RoboDK station: kr30 cnc template half inch flat end mill - paulina 4 AAAAAAAAAAAAAAAAAAAA.rdk

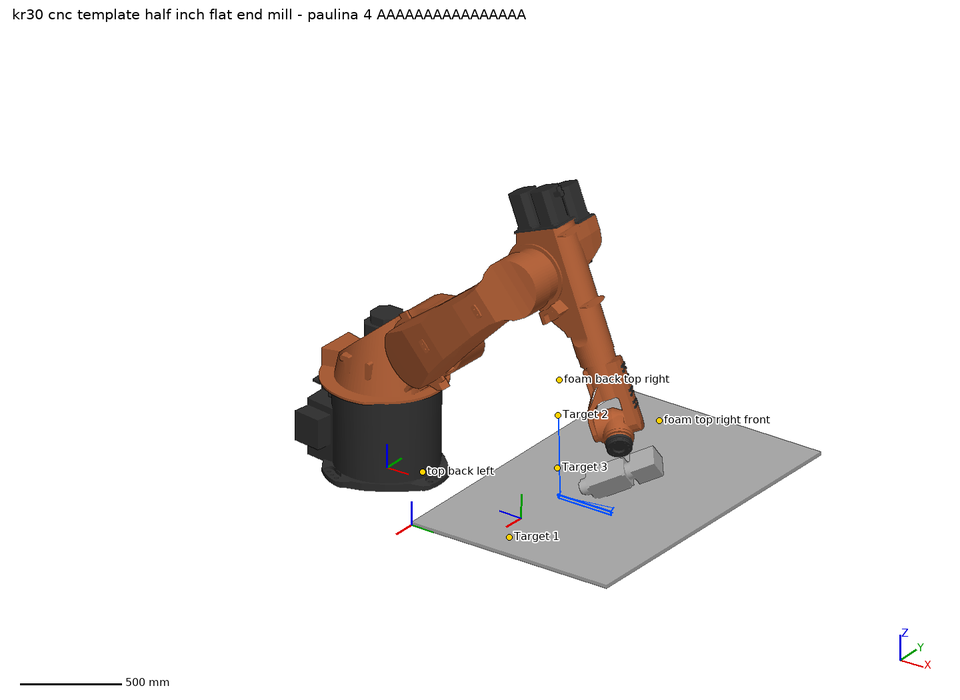
[picture v0: the station drawn from its stored meshes, robots at their saved joint values, targets as dots, program paths as lines]
Station kr30 cnc template half inch flat end mill - paulina 4 AAAAAAAAAAAAAAAAAAAA. Poses are relative to the parent item; angles as X-Y-Z fixed-axis rotations.
  - frame KUKA KR 30 HA Base at (0, 0, 0) mm
    - robot KUKA KR 30 HA: 6 axes, payload 30 kg, reach 2033 mm, repeatability 0.05 mm, weight 665 kg
        modified DH rows (alpha deg, a mm, theta deg, d mm): 0, 0, 0, 815; -90, 350, 0, 0; 0, 850, -90, 0; -90, 145, 0, 820; 90, 0, 0, 0; -90, 0, 180, 170
        joint limits [-185, -135, -120, -350, -119, -350] to [185, 35, 158, 350, 119, 350]; home [0, -90, 90, 0, 0, 0]; saved at [2.296, -41.464, 109.826, -239.674, 53.216, 262.884]
      - tool rc90 spindle mm, TCP at (337.31, -2.2, 160.57) mm, size 110 x 421.3 x 118 mm, geometry from rc90 spindle mm.stl
    - frame Tabletop at (921.82, -1104.91, 385) mm, rotated rx -0.93 ry -0.21 rz -89.9 deg
      - object tabletop CHECK HEIGHT at (-1839.9, 0, 0) mm, size 1839.9 x 1168.4 x 19 mm, geometry from kr30 tabletop mm.stl
      - object kr30 pipe jig base at (-1220, -610.6, 0) mm, size 1217.6 x 88.9 x 88.9 mm, geometry from kr30 pipe jig base.stl
      - frame Frame 3 at (-340, 420, 29) mm, rotated rx 90 ry 0 rz 0 deg
        - target Target 1 (Cartesian target) at (324.46, 69.12, -153.95) mm, rotated rx -179.9 ry 0.14 rz -89.96 deg; joints [37.245, -66.694, 101.534, 53.768, -48.608, -41.204] of KUKA KR 30 HA
        - target Target 2 (Cartesian target) at (-319.2, 432.53, 9.87) mm, rotated rx -179.07 ry 0.05 rz -32.45 deg; joints [8.715, -80.767, 140.791, -170.364, 60.256, 232.965] of KUKA KR 30 HA
        - target Target 3 (Cartesian target) at (-219.35, 204.08, -59.86) mm, rotated rx -178.17 ry 0.56 rz -29.88 deg; joints [13.008, -58.669, 136.899, -167.101, 79.453, 237.713] of KUKA KR 30 HA
    - target foam back top right (Cartesian target) at (1197.65, -230.62, 906.79) mm, rotated rx -15.53 ry 90 rz -15.53 deg; joints [14.757, -102.447, 141.256, 22.791, -41.102, -17.568] of KUKA KR 30 HA
    - target foam top right front (Cartesian target) at (1797.45, -230.62, 850.68) mm, rotated rx -15.58 ry 90 rz -15.58 deg; joints [8.85, -62.405, 99.608, 14.434, -38.093, -11.451] of KUKA KR 30 HA
    - target top back left (Cartesian target) at (1223.08, -1440.01, 894.96) mm, rotated rx 58.97 ry 90 rz 58.97 deg; joints [58.171, -50.232, 76.73, 74.515, -61.834, -59.599] of KUKA KR 30 HA
  - machining project Machining Settings: C:/Users/Research Office/Downloads/b4.apt | rotZ(0) | rotX(0)*rotY(0) | roty(-35) | onStart | onPathStart | onApproach | onPoint | onRetract | onFinish | SetTool(%1) | onPathFinish
  - program Machining (294 instructions, listed below)
  - program Machining (293 instructions, listed below)
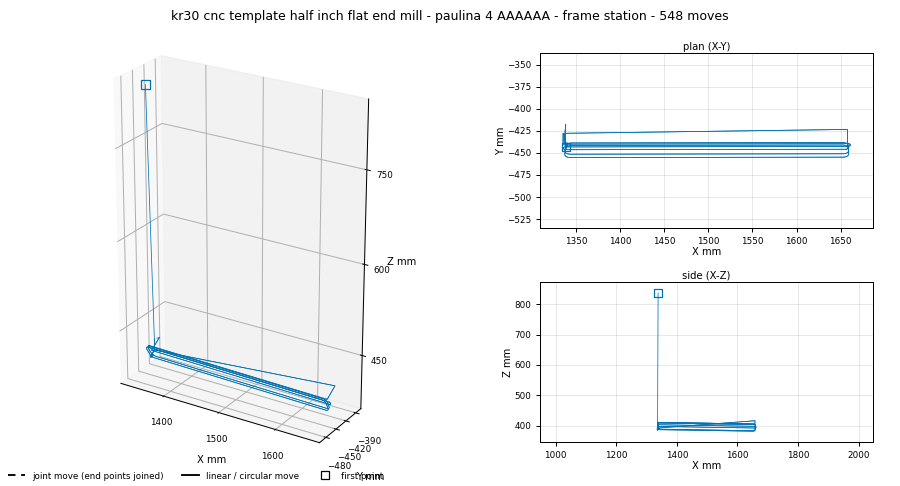
[picture p0: tool path of kr30 cnc template half inch flat end mill - paulina 4 AAAAAAAAAAAAAAAAAAAA.rdk in frame station, 548 of 548 moves have a stored position in this frame; points joined in program order, loops and branches not executed]

--- program Machining (robot KUKA KR 30 HA) ---
  Smooth(10)
  Print: /'1001'
  Print: /''
  Print: /'Contour3'
  Call SetTool(1)
  Set speed (200.0 mm/s)
  Set Ref.: Frame 3
  Set Tool: rc90 spindle mm
  Show rc90 spindle mm
  Set speed (200.0 mm/s)
  MoveJ (Target 2)
  MoveL 619 to (-335.6, -11.85, 4.35) mm, rotated rx -179.15 ry 0 rz -30.08 deg; joints [7.518, -42.725, 139.823, -172.763, 96.85, 241.025]
  MoveL 620 to (-332.9, -13.41, 4.35) mm, rotated rx -179.15 ry 0 rz -30.08 deg; joints [7.669, -42.588, 139.757, -172.61, 96.919, 241.053]
  Set speed (50.0 mm/s)
  MoveL 621 to (-326.98, -16.84, 4.35) mm, rotated rx -179.15 ry 0 rz -30.08 deg; joints [8, -42.287, 139.611, -172.274, 97.068, 241.115]
  MoveL 622 to (-325.36, -16.57, 3.64) mm, rotated rx -179.15 ry 0 rz -30.08 deg; joints [8.085, -42.306, 139.552, -172.19, 96.989, 241.115]
  Set speed (100.0 mm/s)
  MoveL 623 to (-324.39, -14.89, 2.31) mm, rotated rx -179.15 ry 0 rz -30.08 deg; joints [8.128, -42.444, 139.493, -172.15, 96.793, 241.093]
  MoveC 624 to (-324.11, -14.42, 1.33) mm, rotated rx -179.15 ry 0 rz -30.08 deg; joints [8.135, -42.479, 139.434, -172.144, 96.699, 241.081] to (-324.33, -14.8, 0.3) mm, rotated rx -179.15 ry 0 rz -30.08 deg; joints [8.115, -42.44, 139.354, -172.165, 96.659, 241.073]
  MoveL 625 to (-324.33, -14.8, 0.3) mm, rotated rx -179.15 ry 0 rz -30.08 deg; joints [8.115, -42.44, 139.354, -172.165, 96.659, 241.073]
  MoveL 626 to (-324.51, -15.11, -0.05) mm, rotated rx -179.15 ry 0 rz -30.08 deg; joints [8.102, -42.411, 139.324, -172.178, 96.658, 241.071]
  MoveL 627 to (-324.67, -15.38, -0.39) mm, rotated rx -179.15 ry 0 rz -30.08 deg; joints [8.091, -42.385, 139.294, -172.189, 96.654, 241.07]
  MoveL 628 to (-324.81, -15.61, -0.73) mm, rotated rx -179.15 ry 0 rz -30.08 deg; joints [8.081, -42.363, 139.266, -172.2, 96.648, 241.067]
  MoveL 629 to (-324.92, -15.82, -1.07) mm, rotated rx -179.15 ry 0 rz -30.08 deg; joints [8.071, -42.343, 139.237, -172.209, 96.64, 241.065]
  MoveL 630 to (-325.03, -15.99, -1.42) mm, rotated rx -179.15 ry 0 rz -30.08 deg; joints [8.063, -42.326, 139.21, -172.218, 96.63, 241.063]
  MoveL 631 to (-325.11, -16.15, -1.76) mm, rotated rx -179.15 ry 0 rz -30.08 deg; joints [8.055, -42.311, 139.183, -172.225, 96.618, 241.06]
  MoveL 632 to (-325.19, -16.28, -2.1) mm, rotated rx -179.15 ry 0 rz -30.08 deg; joints [8.049, -42.297, 139.156, -172.232, 96.605, 241.058]
  MoveL 633 to (-325.25, -16.39, -2.45) mm, rotated rx -179.15 ry 0 rz -30.08 deg; joints [8.042, -42.285, 139.13, -172.239, 96.591, 241.055]
  MoveL 634 to (-325.31, -16.48, -2.8) mm, rotated rx -179.15 ry 0 rz -30.08 deg; joints [8.037, -42.275, 139.103, -172.245, 96.575, 241.052]
  MoveL 635 to (-325.35, -16.55, -3.14) mm, rotated rx -179.15 ry 0 rz -30.08 deg; joints [8.032, -42.267, 139.077, -172.25, 96.558, 241.049]
  MoveL 636 to (-325.38, -16.61, -3.49) mm, rotated rx -179.15 ry 0 rz -30.08 deg; joints [8.027, -42.26, 139.052, -172.255, 96.54, 241.046]
  MoveL 637 to (-325.41, -16.65, -3.84) mm, rotated rx -179.15 ry 0 rz -30.08 deg; joints [8.023, -42.254, 139.026, -172.26, 96.52, 241.043]
  MoveL 638 to (-325.42, -16.67, -4.19) mm, rotated rx -179.15 ry 0 rz -30.08 deg; joints [8.02, -42.25, 139.001, -172.263, 96.499, 241.04]
  MoveL 639 to (-325.42, -16.68, -4.54) mm, rotated rx -179.15 ry 0 rz -30.08 deg; joints [8.017, -42.247, 138.977, -172.267, 96.478, 241.036]
  MoveL 640 to (-325.42, -16.68, -311.19) mm, rotated rx -179.15 ry 0 rz -30.08 deg; joints [6.155, -36.963, 115.713, -174.061, 78.617, 238.976]
  MoveL 641 to (-325.42, -16.67, -311.54) mm, rotated rx -179.15 ry 0 rz -30.08 deg; joints [6.154, -36.954, 115.684, -174.062, 78.597, 238.974]
  MoveL 642 to (-325.41, -16.65, -311.88) mm, rotated rx -179.15 ry 0 rz -30.08 deg; joints [6.152, -36.946, 115.655, -174.062, 78.577, 238.972]
  MoveL 643 to (-325.38, -16.61, -312.23) mm, rotated rx -179.15 ry 0 rz -30.08 deg; joints [6.152, -36.94, 115.627, -174.063, 78.556, 238.97]
  MoveL 644 to (-325.35, -16.55, -312.58) mm, rotated rx -179.15 ry 0 rz -30.08 deg; joints [6.152, -36.934, 115.599, -174.062, 78.533, 238.968]
  MoveL 645 to (-325.31, -16.48, -312.93) mm, rotated rx -179.15 ry 0 rz -30.08 deg; joints [6.152, -36.93, 115.572, -174.062, 78.51, 238.965]
  MoveL 646 to (-325.25, -16.39, -313.28) mm, rotated rx -179.15 ry 0 rz -30.08 deg; joints [6.152, -36.926, 115.544, -174.061, 78.486, 238.963]
  MoveL 647 to (-325.19, -16.27, -313.63) mm, rotated rx -179.15 ry 0 rz -30.08 deg; joints [6.154, -36.924, 115.517, -174.059, 78.462, 238.96]
  MoveL 648 to (-325.11, -16.14, -313.98) mm, rotated rx -179.15 ry 0 rz -30.08 deg; joints [6.155, -36.923, 115.491, -174.057, 78.436, 238.957]
  MoveL 649 to (-325.02, -15.98, -314.33) mm, rotated rx -179.15 ry 0 rz -30.08 deg; joints [6.157, -36.924, 115.464, -174.054, 78.409, 238.953]
  MoveL 650 to (-324.91, -15.8, -314.68) mm, rotated rx -179.15 ry 0 rz -30.08 deg; joints [6.16, -36.926, 115.438, -174.05, 78.381, 238.95]
  MoveL 651 to (-324.79, -15.59, -315.03) mm, rotated rx -179.15 ry 0 rz -30.08 deg; joints [6.164, -36.93, 115.413, -174.046, 78.352, 238.946]
  MoveL 652 to (-324.65, -15.35, -315.38) mm, rotated rx -179.15 ry 0 rz -30.08 deg; joints [6.168, -36.936, 115.388, -174.041, 78.321, 238.942]
  MoveL 653 to (-324.5, -15.09, -315.7) mm, rotated rx -179.15 ry 0 rz -30.08 deg; joints [6.173, -36.944, 115.365, -174.036, 78.291, 238.938]
  MoveL 654 to (-324.33, -14.8, -316.02) mm, rotated rx -179.15 ry 0 rz -30.08 deg; joints [6.179, -36.954, 115.343, -174.029, 78.259, 238.933]
  MoveL 655 to (-324.16, -14.49, -316.3) mm, rotated rx -179.15 ry 0 rz -30.08 deg; joints [6.185, -36.965, 115.325, -174.022, 78.229, 238.929]
  MoveL 656 to (-323.98, -14.19, -316.55) mm, rotated rx -179.15 ry 0 rz -30.08 deg; joints [6.191, -36.978, 115.309, -174.015, 78.202, 238.924]
  MoveL 657 to (-323.81, -13.89, -316.76) mm, rotated rx -179.15 ry 0 rz -30.08 deg; joints [6.197, -36.991, 115.296, -174.008, 78.176, 238.92]
  MoveL 658 to (-323.63, -13.59, -316.94) mm, rotated rx -179.15 ry 0 rz -30.08 deg; joints [6.204, -37.005, 115.286, -174.001, 78.151, 238.916]
  MoveL 659 to (-323.46, -13.29, -317.1) mm, rotated rx -179.15 ry 0 rz -30.08 deg; joints [6.21, -37.02, 115.277, -173.994, 78.129, 238.913]
  MoveL 660 to (-323.28, -12.99, -317.23) mm, rotated rx -179.15 ry 0 rz -30.08 deg; joints [6.217, -37.036, 115.271, -173.986, 78.107, 238.909]
  MoveL 661 to (-323.11, -12.68, -317.34) mm, rotated rx -179.15 ry 0 rz -30.08 deg; joints [6.224, -37.052, 115.266, -173.979, 78.087, 238.905]
  MoveL 662 to (-322.93, -12.38, -317.43) mm, rotated rx -179.15 ry 0 rz -30.08 deg; joints [6.231, -37.068, 115.264, -173.971, 78.068, 238.902]
  MoveL 663 to (-322.76, -12.08, -317.5) mm, rotated rx -179.15 ry 0 rz -30.08 deg; joints [6.238, -37.085, 115.263, -173.964, 78.05, 238.898]
  MoveL 664 to (-322.58, -11.78, -317.55) mm, rotated rx -179.15 ry 0 rz -30.08 deg; joints [6.245, -37.103, 115.263, -173.956, 78.033, 238.895]
  MoveL 665 to (-322.41, -11.48, -317.58) mm, rotated rx -179.15 ry 0 rz -30.08 deg; joints [6.252, -37.121, 115.266, -173.948, 78.017, 238.892]
  MoveL 666 to (-322.23, -11.17, -317.59) mm, rotated rx -179.15 ry 0 rz -30.08 deg; joints [6.26, -37.14, 115.27, -173.94, 78.003, 238.889]
  MoveL 667 to (-315.94, -0.31, -317.59) mm, rotated rx -179.15 ry 0 rz -30.08 deg; joints [6.525, -37.821, 115.428, -173.657, 77.489, 238.774]
  MoveL 668 to (-315.59, 0.29, -317.58) mm, rotated rx -179.15 ry 0 rz -30.08 deg; joints [6.54, -37.859, 115.438, -173.641, 77.461, 238.768]
  MoveL 669 to (-315.42, 0.6, -317.55) mm, rotated rx -179.15 ry 0 rz -30.08 deg; joints [6.547, -37.879, 115.444, -173.633, 77.448, 238.765]
  MoveL 670 to (-315.24, 0.9, -317.5) mm, rotated rx -179.15 ry 0 rz -30.08 deg; joints [6.555, -37.899, 115.452, -173.625, 77.437, 238.762]
  MoveL 671 to (-315.07, 1.2, -317.43) mm, rotated rx -179.15 ry 0 rz -30.08 deg; joints [6.562, -37.92, 115.462, -173.617, 77.426, 238.759]
  MoveL 672 to (-314.89, 1.5, -317.34) mm, rotated rx -179.15 ry 0 rz -30.08 deg; joints [6.57, -37.941, 115.474, -173.609, 77.416, 238.756]
  MoveL 673 to (-314.72, 1.8, -317.23) mm, rotated rx -179.15 ry 0 rz -30.08 deg; joints [6.578, -37.963, 115.487, -173.6, 77.408, 238.753]
  MoveL 674 to (-314.54, 2.1, -317.1) mm, rotated rx -179.15 ry 0 rz -30.08 deg; joints [6.586, -37.986, 115.502, -173.592, 77.401, 238.75]
  MoveL 675 to (-314.39, 2.36, -316.97) mm, rotated rx -179.15 ry 0 rz -30.08 deg; joints [6.593, -38.005, 115.517, -173.585, 77.396, 238.748]
  MoveL 676 to (-314.24, 2.62, -316.82) mm, rotated rx -179.15 ry 0 rz -30.08 deg; joints [6.6, -38.026, 115.533, -173.577, 77.392, 238.746]
  MoveL 677 to (-314.09, 2.88, -316.65) mm, rotated rx -179.15 ry 0 rz -30.08 deg; joints [6.607, -38.047, 115.551, -173.57, 77.389, 238.744]
  MoveL 678 to (-313.95, 3.13, -316.45) mm, rotated rx -179.15 ry 0 rz -30.08 deg; joints [6.614, -38.068, 115.57, -173.563, 77.387, 238.743]
  MoveL 679 to (-313.8, 3.39, -316.23) mm, rotated rx -179.15 ry 0 rz -30.08 deg; joints [6.622, -38.09, 115.592, -173.555, 77.387, 238.741]
  MoveL 680 to (-313.65, 3.65, -315.98) mm, rotated rx -179.15 ry 0 rz -30.08 deg; joints [6.629, -38.113, 115.616, -173.547, 77.388, 238.739]
  MoveL 681 to (-313.49, 3.92, -315.68) mm, rotated rx -179.15 ry 0 rz -30.08 deg; joints [6.638, -38.139, 115.645, -173.539, 77.392, 238.738]
  MoveL 682 to (-313.35, 4.16, -315.38) mm, rotated rx -179.15 ry 0 rz -30.08 deg; joints [6.645, -38.162, 115.673, -173.532, 77.397, 238.737]
  MoveL 683 to (-313.24, 4.35, -315.11) mm, rotated rx -179.15 ry 0 rz -30.08 deg; joints [6.651, -38.181, 115.698, -173.526, 77.402, 238.736]
  MoveL 684 to (-313.14, 4.52, -314.85) mm, rotated rx -179.15 ry 0 rz -30.08 deg; joints [6.656, -38.199, 115.722, -173.52, 77.409, 238.736]
  MoveL 685 to (-313.05, 4.68, -314.57) mm, rotated rx -179.15 ry 0 rz -30.08 deg; joints [6.662, -38.217, 115.747, -173.515, 77.416, 238.735]
  MoveL 686 to (-312.97, 4.82, -314.28) mm, rotated rx -179.15 ry 0 rz -30.08 deg; joints [6.666, -38.234, 115.773, -173.51, 77.425, 238.735]
  MoveL 687 to (-312.9, 4.95, -314) mm, rotated rx -179.15 ry 0 rz -30.08 deg; joints [6.671, -38.249, 115.798, -173.506, 77.435, 238.735]
  MoveL 688 to (-312.83, 5.06, -313.72) mm, rotated rx -179.15 ry 0 rz -30.08 deg; joints [6.675, -38.264, 115.823, -173.502, 77.445, 238.736]
  MoveL 689 to (-312.73, 5.24, -313.15) mm, rotated rx -179.15 ry 0 rz -30.08 deg; joints [6.682, -38.291, 115.872, -173.495, 77.467, 238.737]
  MoveL 690 to (-312.65, 5.37, -312.58) mm, rotated rx -179.15 ry 0 rz -30.08 deg; joints [6.688, -38.315, 115.92, -173.489, 77.492, 238.738]
  MoveL 691 to (-312.62, 5.43, -312.23) mm, rotated rx -179.15 ry 0 rz -30.08 deg; joints [6.692, -38.328, 115.95, -173.486, 77.508, 238.739]
  MoveL 692 to (-312.59, 5.47, -311.88) mm, rotated rx -179.15 ry 0 rz -30.08 deg; joints [6.694, -38.34, 115.979, -173.484, 77.525, 238.741]
  MoveL 693 to (-312.58, 5.49, -311.54) mm, rotated rx -179.15 ry 0 rz -30.08 deg; joints [6.697, -38.351, 116.009, -173.482, 77.543, 238.742]
  MoveL 694 to (-312.58, 5.49, -311.19) mm, rotated rx -179.15 ry 0 rz -30.08 deg; joints [6.699, -38.361, 116.037, -173.481, 77.562, 238.744]
  MoveL 695 to (-312.58, 5.49, -5.24) mm, rotated rx -179.15 ry 0 rz -30.08 deg; joints [8.711, -44.154, 139.346, -171.59, 94.945, 240.891]
  MoveL 696 to (-312.58, 5.49, -2.45) mm, rotated rx -179.15 ry 0 rz -30.08 deg; joints [8.735, -44.177, 139.543, -171.564, 95.117, 240.919]
  MoveL 697 to (-312.59, 5.47, -2.1) mm, rotated rx -179.15 ry 0 rz -30.08 deg; joints [8.737, -44.178, 139.568, -171.562, 95.14, 240.923]
  MoveL 698 to (-312.62, 5.43, -1.75) mm, rotated rx -179.15 ry 0 rz -30.08 deg; joints [8.739, -44.178, 139.592, -171.56, 95.164, 240.926]
  MoveL 699 to (-312.65, 5.37, -1.4) mm, rotated rx -179.15 ry 0 rz -30.08 deg; joints [8.74, -44.176, 139.615, -171.558, 95.19, 240.93]
  MoveL 700 to (-312.69, 5.3, -1.05) mm, rotated rx -179.15 ry 0 rz -30.08 deg; joints [8.741, -44.172, 139.639, -171.557, 95.216, 240.934]
  MoveL 701 to (-312.75, 5.2, -0.7) mm, rotated rx -179.15 ry 0 rz -30.08 deg; joints [8.741, -44.167, 139.662, -171.557, 95.244, 240.938]
  MoveL 702 to (-312.81, 5.09, -0.35) mm, rotated rx -179.15 ry 0 rz -30.08 deg; joints [8.74, -44.16, 139.684, -171.557, 95.273, 240.943]
  MoveL 703 to (-312.89, 4.96, 0) mm, rotated rx -179.15 ry 0 rz -30.08 deg; joints [8.739, -44.152, 139.707, -171.558, 95.304, 240.947]
  MoveL 704 to (-312.98, 4.8, 0.35) mm, rotated rx -179.15 ry 0 rz -30.08 deg; joints [8.737, -44.141, 139.728, -171.559, 95.336, 240.952]
  MoveL 705 to (-313.06, 4.67, 0.61) mm, rotated rx -179.15 ry 0 rz -30.08 deg; joints [8.735, -44.131, 139.745, -171.561, 95.362, 240.955]
  MoveL 706 to (-313.14, 4.52, 0.87) mm, rotated rx -179.15 ry 0 rz -30.08 deg; joints [8.733, -44.121, 139.76, -171.563, 95.388, 240.959]
  MoveL 707 to (-313.28, 4.28, 1.23) mm, rotated rx -179.15 ry 0 rz -30.08 deg; joints [8.728, -44.103, 139.782, -171.567, 95.426, 240.964]
  MoveL 708 to (-313.44, 4.01, 1.6) mm, rotated rx -179.15 ry 0 rz -30.08 deg; joints [8.723, -44.082, 139.802, -171.572, 95.468, 240.97]
  MoveL 709 to (-313.54, 3.84, 1.8) mm, rotated rx -179.15 ry 0 rz -30.08 deg; joints [8.719, -44.069, 139.814, -171.575, 95.492, 240.973]
  MoveL 710 to (-313.64, 3.66, 1.99) mm, rotated rx -179.15 ry 0 rz -30.08 deg; joints [8.715, -44.055, 139.824, -171.579, 95.516, 240.976]
  MoveL 711 to (-313.84, 3.31, 2.32) mm, rotated rx -179.15 ry 0 rz -30.08 deg; joints [8.707, -44.027, 139.841, -171.586, 95.561, 240.982]
  MoveL 712 to (-314.02, 3.01, 2.57) mm, rotated rx -179.15 ry 0 rz -30.08 deg; joints [8.699, -44.003, 139.853, -171.593, 95.597, 240.987]
  MoveL 713 to (-314.19, 2.71, 2.78) mm, rotated rx -179.15 ry 0 rz -30.08 deg; joints [8.691, -43.978, 139.863, -171.601, 95.63, 240.991]
  MoveL 714 to (-314.37, 2.41, 2.96) mm, rotated rx -179.15 ry 0 rz -30.08 deg; joints [8.683, -43.953, 139.87, -171.608, 95.663, 240.995]
  MoveL 715 to (-314.54, 2.1, 3.12) mm, rotated rx -179.15 ry 0 rz -30.08 deg; joints [8.675, -43.928, 139.876, -171.616, 95.693, 240.998]
  MoveL 716 to (-314.57, 2.06, 3.14) mm, rotated rx -179.15 ry 0 rz -30.08 deg; joints [8.674, -43.925, 139.876, -171.617, 95.697, 240.999]
  MoveL 717 to (-314.74, 1.76, 3.27) mm, rotated rx -179.15 ry 0 rz -30.08 deg; joints [8.666, -43.9, 139.88, -171.625, 95.725, 241.002]
  MoveL 718 to (-314.91, 1.47, 3.37) mm, rotated rx -179.15 ry 0 rz -30.08 deg; joints [8.657, -43.875, 139.882, -171.633, 95.752, 241.005]
  MoveL 719 to (-315.08, 1.17, 3.46) mm, rotated rx -179.15 ry 0 rz -30.08 deg; joints [8.648, -43.85, 139.882, -171.642, 95.778, 241.008]
  MoveL 720 to (-315.25, 0.88, 3.52) mm, rotated rx -179.15 ry 0 rz -30.08 deg; joints [8.64, -43.824, 139.882, -171.65, 95.802, 241.011]
  MoveL 721 to (-315.43, 0.58, 3.57) mm, rotated rx -179.15 ry 0 rz -30.08 deg; joints [8.631, -43.799, 139.879, -171.659, 95.826, 241.013]
  MoveL 722 to (-315.6, 0.28, 3.6) mm, rotated rx -179.15 ry 0 rz -30.08 deg; joints [8.621, -43.773, 139.876, -171.668, 95.848, 241.016]
  MoveL 723 to (-315.94, -0.31, 3.61) mm, rotated rx -179.15 ry 0 rz -30.08 deg; joints [8.603, -43.722, 139.866, -171.686, 95.889, 241.02]
  MoveL 724 to (-316.64, -1.52, 3.61) mm, rotated rx -179.15 ry 0 rz -30.08 deg; joints [8.564, -43.616, 139.843, -171.724, 95.971, 241.027]
  MoveL 725 to (-316.99, -2.12, 3.58) mm, rotated rx -179.15 ry 0 rz -30.08 deg; joints [8.545, -43.564, 139.83, -171.742, 96.011, 241.031]
  MoveL 726 to (-317.34, -2.72, 3.49) mm, rotated rx -179.15 ry 0 rz -30.08 deg; joints [8.525, -43.51, 139.813, -171.762, 96.047, 241.034]
  MoveL 727 to (-321.53, -9.97, 2.16) mm, rotated rx -179.15 ry 0 rz -30.08 deg; joints [8.283, -42.871, 139.581, -171.998, 96.454, 241.065]
  MoveL 728 to (-322.93, -12.38, 1.71) mm, rotated rx -179.15 ry 0 rz -30.08 deg; joints [8.203, -42.658, 139.501, -172.077, 96.587, 241.074]
  MoveL 729 to (-323.1, -12.68, 1.62) mm, rotated rx -179.15 ry 0 rz -30.08 deg; joints [8.193, -42.632, 139.49, -172.087, 96.602, 241.075]
  MoveL 730 to (-323.28, -12.97, 1.52) mm, rotated rx -179.15 ry 0 rz -30.08 deg; joints [8.183, -42.606, 139.476, -172.097, 96.615, 241.075]
  MoveL 731 to (-323.45, -13.27, 1.39) mm, rotated rx -179.15 ry 0 rz -30.08 deg; joints [8.172, -42.579, 139.461, -172.108, 96.626, 241.076]
  MoveL 732 to (-323.62, -13.56, 1.24) mm, rotated rx -179.15 ry 0 rz -30.08 deg; joints [8.161, -42.553, 139.445, -172.118, 96.636, 241.076]
  MoveL 733 to (-323.79, -13.86, 1.06) mm, rotated rx -179.15 ry 0 rz -30.08 deg; joints [8.151, -42.526, 139.426, -172.129, 96.645, 241.076]
  MoveL 734 to (-323.96, -14.15, 0.85) mm, rotated rx -179.15 ry 0 rz -30.08 deg; joints [8.14, -42.499, 139.406, -172.14, 96.652, 241.075]
  MoveL 735 to (-324.13, -14.45, 0.62) mm, rotated rx -179.15 ry 0 rz -30.08 deg; joints [8.128, -42.472, 139.384, -172.151, 96.656, 241.074]
  MoveL 736 to (-324.3, -14.75, 0.35) mm, rotated rx -179.15 ry 0 rz -30.08 deg; joints [8.117, -42.445, 139.359, -172.163, 96.659, 241.073]
  MoveL 737 to (-324.33, -14.8, 0.3) mm, rotated rx -179.15 ry 0 rz -30.08 deg; joints [8.115, -42.44, 139.354, -172.165, 96.659, 241.073]
  MoveC 738 to (-325.22, -16.33, 0.41) mm, rotated rx -179.15 ry 0 rz -30.08 deg; joints [8.067, -42.308, 139.331, -172.211, 96.768, 241.082] to (-325.18, -16.27, 2.18) mm, rotated rx -179.15 ry 0 rz -30.08 deg; joints [8.083, -42.323, 139.456, -172.193, 96.876, 241.099]
  MoveL 739 to (-325.18, -16.27, 2.18) mm, rotated rx -179.15 ry 0 rz -30.08 deg; joints [8.083, -42.323, 139.456, -172.193, 96.876, 241.099]
  MoveL 740 to (-324.74, -15.51, 3.02) mm, rotated rx -179.15 ry 0 rz -30.08 deg; joints [8.114, -42.395, 139.53, -172.162, 96.879, 241.103]
  Set speed (50.0 mm/s)
  MoveL 741 to (-322.97, -16.53, 3.02) mm, rotated rx -179.15 ry 0 rz -30.08 deg; joints [8.213, -42.305, 139.486, -172.062, 96.922, 241.122]
  MoveL 742 to (-321.44, -16.41, 2.09) mm, rotated rx -179.15 ry 0 rz -30.08 deg; joints [8.29, -42.309, 139.409, -171.985, 96.84, 241.12]
  Set speed (100.0 mm/s)
  MoveC 743 to (-321.26, -16.11, 1.18) mm, rotated rx -179.15 ry 0 rz -30.08 deg; joints [8.293, -42.33, 139.351, -171.984, 96.762, 241.11] to (-321.46, -16.46, 0.3) mm, rotated rx -179.15 ry 0 rz -30.08 deg; joints [8.274, -42.295, 139.282, -172.003, 96.729, 241.103]
  MoveL 744 to (-321.46, -16.46, 0.3) mm, rotated rx -179.15 ry 0 rz -30.08 deg; joints [8.274, -42.295, 139.282, -172.003, 96.729, 241.103]
  MoveL 745 to (-321.65, -16.77, -0.05) mm, rotated rx -179.15 ry 0 rz -30.08 deg; joints [8.262, -42.265, 139.252, -172.016, 96.728, 241.101]
  MoveL 746 to (-321.8, -17.04, -0.39) mm, rotated rx -179.15 ry 0 rz -30.08 deg; joints [8.25, -42.24, 139.222, -172.028, 96.724, 241.099]
  MoveL 747 to (-321.94, -17.28, -0.73) mm, rotated rx -179.15 ry 0 rz -30.08 deg; joints [8.24, -42.218, 139.194, -172.038, 96.718, 241.097]
  MoveL 748 to (-322.05, -17.48, -1.07) mm, rotated rx -179.15 ry 0 rz -30.08 deg; joints [8.231, -42.198, 139.166, -172.047, 96.71, 241.094]
  MoveL 749 to (-322.16, -17.66, -1.42) mm, rotated rx -179.15 ry 0 rz -30.08 deg; joints [8.222, -42.181, 139.138, -172.056, 96.7, 241.092]
  MoveL 750 to (-322.25, -17.81, -1.76) mm, rotated rx -179.15 ry 0 rz -30.08 deg; joints [8.215, -42.166, 139.111, -172.064, 96.688, 241.089]
  MoveL 751 to (-322.32, -17.94, -2.1) mm, rotated rx -179.15 ry 0 rz -30.08 deg; joints [8.208, -42.152, 139.084, -172.071, 96.675, 241.087]
  MoveL 752 to (-322.38, -18.05, -2.45) mm, rotated rx -179.15 ry 0 rz -30.08 deg; joints [8.202, -42.141, 139.058, -172.078, 96.661, 241.084]
  MoveL 753 to (-322.44, -18.14, -2.8) mm, rotated rx -179.15 ry 0 rz -30.08 deg; joints [8.196, -42.13, 139.032, -172.084, 96.645, 241.081]
  MoveL 754 to (-322.48, -18.22, -3.14) mm, rotated rx -179.15 ry 0 rz -30.08 deg; joints [8.191, -42.122, 139.006, -172.089, 96.628, 241.078]
  MoveL 755 to (-322.51, -18.27, -3.49) mm, rotated rx -179.15 ry 0 rz -30.08 deg; joints [8.186, -42.115, 138.98, -172.094, 96.609, 241.075]
  MoveL 756 to (-322.54, -18.31, -3.84) mm, rotated rx -179.15 ry 0 rz -30.08 deg; joints [8.182, -42.109, 138.955, -172.098, 96.59, 241.072]
  MoveL 757 to (-322.55, -18.34, -4.19) mm, rotated rx -179.15 ry 0 rz -30.08 deg; joints [8.179, -42.105, 138.93, -172.102, 96.569, 241.068]
  MoveL 758 to (-322.55, -18.34, -4.54) mm, rotated rx -179.15 ry 0 rz -30.08 deg; joints [8.176, -42.102, 138.905, -172.106, 96.548, 241.065]
  MoveL 759 to (-322.55, -18.34, -311.19) mm, rotated rx -179.15 ry 0 rz -30.08 deg; joints [6.278, -36.848, 115.652, -173.936, 78.674, 238.958]
  MoveL 760 to (-322.55, -18.33, -311.54) mm, rotated rx -179.15 ry 0 rz -30.08 deg; joints [6.277, -36.839, 115.623, -173.937, 78.654, 238.956]
  MoveL 761 to (-322.54, -18.31, -311.88) mm, rotated rx -179.15 ry 0 rz -30.08 deg; joints [6.275, -36.831, 115.595, -173.938, 78.633, 238.954]
  MoveL 762 to (-322.51, -18.27, -312.23) mm, rotated rx -179.15 ry 0 rz -30.08 deg; joints [6.275, -36.825, 115.567, -173.938, 78.612, 238.952]
  MoveL 763 to (-322.48, -18.22, -312.58) mm, rotated rx -179.15 ry 0 rz -30.08 deg; joints [6.275, -36.819, 115.539, -173.938, 78.59, 238.949]
  MoveL 764 to (-322.44, -18.14, -312.93) mm, rotated rx -179.15 ry 0 rz -30.08 deg; joints [6.275, -36.815, 115.511, -173.938, 78.567, 238.947]
  MoveL 765 to (-322.38, -18.05, -313.28) mm, rotated rx -179.15 ry 0 rz -30.08 deg; joints [6.275, -36.811, 115.484, -173.936, 78.543, 238.944]
  MoveL 766 to (-322.32, -17.93, -313.63) mm, rotated rx -179.15 ry 0 rz -30.08 deg; joints [6.276, -36.809, 115.457, -173.935, 78.518, 238.941]
  MoveL 767 to (-322.24, -17.8, -313.98) mm, rotated rx -179.15 ry 0 rz -30.08 deg; joints [6.278, -36.809, 115.43, -173.933, 78.492, 238.938]
  MoveL 768 to (-322.15, -17.64, -314.33) mm, rotated rx -179.15 ry 0 rz -30.08 deg; joints [6.28, -36.809, 115.404, -173.93, 78.466, 238.935]
  MoveL 769 to (-322.05, -17.46, -314.68) mm, rotated rx -179.15 ry 0 rz -30.08 deg; joints [6.283, -36.811, 115.378, -173.926, 78.438, 238.931]
  MoveL 770 to (-321.92, -17.25, -315.03) mm, rotated rx -179.15 ry 0 rz -30.08 deg; joints [6.286, -36.815, 115.352, -173.922, 78.408, 238.927]
  MoveL 771 to (-321.78, -17.01, -315.38) mm, rotated rx -179.15 ry 0 rz -30.08 deg; joints [6.291, -36.821, 115.327, -173.917, 78.378, 238.923]
  MoveL 772 to (-321.63, -16.75, -315.7) mm, rotated rx -179.15 ry 0 rz -30.08 deg; joints [6.295, -36.829, 115.305, -173.912, 78.348, 238.919]
  MoveL 773 to (-321.46, -16.46, -316.02) mm, rotated rx -179.15 ry 0 rz -30.08 deg; joints [6.301, -36.839, 115.283, -173.905, 78.316, 238.914]
  MoveL 774 to (-321.29, -16.16, -316.3) mm, rotated rx -179.15 ry 0 rz -30.08 deg; joints [6.307, -36.851, 115.264, -173.898, 78.286, 238.909]
  MoveL 775 to (-321.11, -15.85, -316.55) mm, rotated rx -179.15 ry 0 rz -30.08 deg; joints [6.313, -36.863, 115.248, -173.891, 78.258, 238.905]
  MoveL 776 to (-320.94, -15.55, -316.76) mm, rotated rx -179.15 ry 0 rz -30.08 deg; joints [6.32, -36.877, 115.236, -173.884, 78.232, 238.901]
  MoveL 777 to (-320.76, -15.25, -316.94) mm, rotated rx -179.15 ry 0 rz -30.08 deg; joints [6.326, -36.891, 115.225, -173.877, 78.208, 238.897]
  MoveL 778 to (-320.59, -14.95, -317.1) mm, rotated rx -179.15 ry 0 rz -30.08 deg; joints [6.333, -36.905, 115.217, -173.87, 78.185, 238.893]
  MoveL 779 to (-320.41, -14.65, -317.23) mm, rotated rx -179.15 ry 0 rz -30.08 deg; joints [6.34, -36.921, 115.21, -173.862, 78.164, 238.889]
  MoveL 780 to (-320.24, -14.35, -317.34) mm, rotated rx -179.15 ry 0 rz -30.08 deg; joints [6.346, -36.937, 115.206, -173.855, 78.143, 238.886]
  MoveL 781 to (-320.06, -14.04, -317.43) mm, rotated rx -179.15 ry 0 rz -30.08 deg; joints [6.353, -36.954, 115.203, -173.847, 78.124, 238.882]
  MoveL 782 to (-319.89, -13.74, -317.5) mm, rotated rx -179.15 ry 0 rz -30.08 deg; joints [6.36, -36.971, 115.202, -173.84, 78.106, 238.879]
  MoveL 783 to (-319.71, -13.44, -317.55) mm, rotated rx -179.15 ry 0 rz -30.08 deg; joints [6.368, -36.988, 115.203, -173.832, 78.09, 238.875]
  MoveL 784 to (-319.54, -13.14, -317.58) mm, rotated rx -179.15 ry 0 rz -30.08 deg; joints [6.375, -37.007, 115.205, -173.824, 78.074, 238.872]
  MoveL 785 to (-319.37, -12.84, -317.59) mm, rotated rx -179.15 ry 0 rz -30.08 deg; joints [6.382, -37.025, 115.209, -173.817, 78.059, 238.869]
  MoveL 786 to (-312.02, -0.16, -317.59) mm, rotated rx -179.15 ry 0 rz -30.08 deg; joints [6.691, -37.82, 115.394, -173.486, 77.461, 238.734]
  MoveL 787 to (-311.85, 0.14, -317.58) mm, rotated rx -179.15 ry 0 rz -30.08 deg; joints [6.699, -37.839, 115.398, -173.478, 77.446, 238.731]
  MoveL 788 to (-311.67, 0.44, -317.56) mm, rotated rx -179.15 ry 0 rz -30.08 deg; joints [6.706, -37.858, 115.404, -173.47, 77.433, 238.727]
  MoveL 789 to (-311.5, 0.74, -317.53) mm, rotated rx -179.15 ry 0 rz -30.08 deg; joints [6.714, -37.878, 115.411, -173.462, 77.421, 238.724]
  MoveL 790 to (-311.32, 1.05, -317.47) mm, rotated rx -179.15 ry 0 rz -30.08 deg; joints [6.721, -37.898, 115.42, -173.454, 77.409, 238.721]
  MoveL 791 to (-311.15, 1.35, -317.39) mm, rotated rx -179.15 ry 0 rz -30.08 deg; joints [6.729, -37.919, 115.431, -173.445, 77.399, 238.718]
  MoveL 792 to (-310.97, 1.65, -317.29) mm, rotated rx -179.15 ry 0 rz -30.08 deg; joints [6.737, -37.941, 115.443, -173.437, 77.39, 238.716]
  MoveL 793 to (-310.8, 1.95, -317.17) mm, rotated rx -179.15 ry 0 rz -30.08 deg; joints [6.745, -37.963, 115.457, -173.429, 77.382, 238.713]
  MoveL 794 to (-310.62, 2.25, -317.03) mm, rotated rx -179.15 ry 0 rz -30.08 deg; joints [6.753, -37.986, 115.473, -173.42, 77.376, 238.71]
  MoveL 795 to (-310.45, 2.55, -316.86) mm, rotated rx -179.15 ry 0 rz -30.08 deg; joints [6.761, -38.009, 115.491, -173.412, 77.371, 238.708]
  MoveL 796 to (-310.28, 2.86, -316.66) mm, rotated rx -179.15 ry 0 rz -30.08 deg; joints [6.769, -38.034, 115.512, -173.403, 77.367, 238.706]
  MoveL 797 to (-310.09, 3.18, -316.41) mm, rotated rx -179.15 ry 0 rz -30.08 deg; joints [6.779, -38.061, 115.537, -173.394, 77.365, 238.703]
  MoveL 798 to (-309.9, 3.51, -316.12) mm, rotated rx -179.15 ry 0 rz -30.08 deg; joints [6.788, -38.09, 115.565, -173.384, 77.365, 238.701]
  MoveL 799 to (-309.71, 3.84, -315.78) mm, rotated rx -179.15 ry 0 rz -30.08 deg; joints [6.798, -38.119, 115.598, -173.374, 77.368, 238.699]
  MoveL 800 to (-309.52, 4.16, -315.38) mm, rotated rx -179.15 ry 0 rz -30.08 deg; joints [6.808, -38.151, 115.636, -173.364, 77.375, 238.698]
  MoveL 801 to (-309.4, 4.37, -315.08) mm, rotated rx -179.15 ry 0 rz -30.08 deg; joints [6.814, -38.172, 115.663, -173.357, 77.381, 238.697]
  MoveL 802 to (-309.29, 4.55, -314.79) mm, rotated rx -179.15 ry 0 rz -30.08 deg; joints [6.82, -38.191, 115.689, -173.351, 77.388, 238.697]
  MoveL 803 to (-309.2, 4.71, -314.5) mm, rotated rx -179.15 ry 0 rz -30.08 deg; joints [6.826, -38.21, 115.716, -173.346, 77.396, 238.696]
  MoveL 804 to (-309.12, 4.86, -314.2) mm, rotated rx -179.15 ry 0 rz -30.08 deg; joints [6.831, -38.227, 115.742, -173.341, 77.406, 238.696]
  MoveL 805 to (-309.04, 4.98, -313.91) mm, rotated rx -179.15 ry 0 rz -30.08 deg; joints [6.835, -38.243, 115.768, -173.337, 77.416, 238.697]
  MoveL 806 to (-308.98, 5.09, -313.62) mm, rotated rx -179.15 ry 0 rz -30.08 deg; joints [6.84, -38.258, 115.794, -173.333, 77.426, 238.697]
  MoveL 807 to (-308.88, 5.27, -313.03) mm, rotated rx -179.15 ry 0 rz -30.08 deg; joints [6.847, -38.285, 115.845, -173.326, 77.45, 238.698]
  MoveL 808 to (-308.82, 5.37, -312.58) mm, rotated rx -179.15 ry 0 rz -30.08 deg; joints [6.852, -38.304, 115.883, -173.321, 77.47, 238.699]
  MoveL 809 to (-308.79, 5.43, -312.23) mm, rotated rx -179.15 ry 0 rz -30.08 deg; joints [6.855, -38.317, 115.912, -173.319, 77.486, 238.701]
  MoveL 810 to (-308.76, 5.47, -311.88) mm, rotated rx -179.15 ry 0 rz -30.08 deg; joints [6.858, -38.329, 115.942, -173.316, 77.503, 238.702]
  MoveL 811 to (-308.75, 5.49, -311.54) mm, rotated rx -179.15 ry 0 rz -30.08 deg; joints [6.86, -38.34, 115.971, -173.314, 77.521, 238.704]
  MoveL 812 to (-308.75, 5.49, -311.19) mm, rotated rx -179.15 ry 0 rz -30.08 deg; joints [6.862, -38.35, 116, -173.313, 77.54, 238.706]
  MoveL 813 to (-308.75, 5.49, -5.24) mm, rotated rx -179.15 ry 0 rz -30.08 deg; joints [8.922, -44.151, 139.304, -171.38, 94.904, 240.904]
  MoveL 814 to (-308.75, 5.49, -2.45) mm, rotated rx -179.15 ry 0 rz -30.08 deg; joints [8.946, -44.174, 139.502, -171.353, 95.076, 240.933]
  MoveL 815 to (-308.76, 5.46, -2.07) mm, rotated rx -179.15 ry 0 rz -30.08 deg; joints [8.948, -44.175, 139.527, -171.35, 95.1, 240.937]
  MoveL 816 to (-308.79, 5.42, -1.7) mm, rotated rx -179.15 ry 0 rz -30.08 deg; joints [8.95, -44.175, 139.553, -171.348, 95.126, 240.941]
  MoveL 817 to (-308.83, 5.36, -1.32) mm, rotated rx -179.15 ry 0 rz -30.08 deg; joints [8.951, -44.172, 139.578, -171.346, 95.154, 240.945]
  MoveL 818 to (-308.88, 5.27, -0.95) mm, rotated rx -179.15 ry 0 rz -30.08 deg; joints [8.952, -44.168, 139.603, -171.345, 95.182, 240.95]
  MoveL 819 to (-308.93, 5.18, -0.63) mm, rotated rx -179.15 ry 0 rz -30.08 deg; joints [8.952, -44.163, 139.625, -171.345, 95.209, 240.954]
  MoveL 820 to (-308.99, 5.07, -0.3) mm, rotated rx -179.15 ry 0 rz -30.08 deg; joints [8.951, -44.156, 139.646, -171.345, 95.236, 240.958]
  MoveL 821 to (-309.06, 4.95, 0.02) mm, rotated rx -179.15 ry 0 rz -30.08 deg; joints [8.95, -44.148, 139.666, -171.346, 95.265, 240.962]
  MoveL 822 to (-309.15, 4.8, 0.35) mm, rotated rx -179.15 ry 0 rz -30.08 deg; joints [8.949, -44.138, 139.687, -171.347, 95.295, 240.966]
  MoveL 823 to (-309.24, 4.65, 0.64) mm, rotated rx -179.15 ry 0 rz -30.08 deg; joints [8.946, -44.127, 139.705, -171.349, 95.323, 240.97]
  MoveL 824 to (-309.33, 4.48, 0.93) mm, rotated rx -179.15 ry 0 rz -30.08 deg; joints [8.944, -44.115, 139.722, -171.351, 95.352, 240.975]
  MoveL 825 to (-309.44, 4.29, 1.22) mm, rotated rx -179.15 ry 0 rz -30.08 deg; joints [8.94, -44.101, 139.739, -171.354, 95.383, 240.979]
  MoveL 826 to (-309.57, 4.08, 1.51) mm, rotated rx -179.15 ry 0 rz -30.08 deg; joints [8.936, -44.085, 139.756, -171.358, 95.416, 240.984]
  MoveL 827 to (-309.75, 3.77, 1.87) mm, rotated rx -179.15 ry 0 rz -30.08 deg; joints [8.929, -44.061, 139.776, -171.364, 95.459, 240.99]
  MoveL 828 to (-309.92, 3.47, 2.18) mm, rotated rx -179.15 ry 0 rz -30.08 deg; joints [8.922, -44.037, 139.792, -171.37, 95.499, 240.995]
  MoveL 829 to (-310.1, 3.16, 2.45) mm, rotated rx -179.15 ry 0 rz -30.08 deg; joints [8.915, -44.013, 139.806, -171.377, 95.537, 241]
  MoveL 830 to (-310.27, 2.86, 2.68) mm, rotated rx -179.15 ry 0 rz -30.08 deg; joints [8.907, -43.988, 139.817, -171.384, 95.572, 241.005]
  MoveL 831 to (-310.39, 2.66, 2.81) mm, rotated rx -179.15 ry 0 rz -30.08 deg; joints [8.902, -43.972, 139.822, -171.389, 95.594, 241.007]
  MoveL 832 to (-310.51, 2.46, 2.93) mm, rotated rx -179.15 ry 0 rz -30.08 deg; joints [8.897, -43.955, 139.827, -171.394, 95.615, 241.01]
  MoveL 833 to (-310.74, 2.06, 3.14) mm, rotated rx -179.15 ry 0 rz -30.08 deg; joints [8.886, -43.922, 139.835, -171.404, 95.655, 241.015]
  MoveL 834 to (-310.97, 1.66, 3.31) mm, rotated rx -179.15 ry 0 rz -30.08 deg; joints [8.875, -43.888, 139.839, -171.415, 95.694, 241.02]
  MoveL 835 to (-311.2, 1.25, 3.44) mm, rotated rx -179.15 ry 0 rz -30.08 deg; joints [8.863, -43.854, 139.841, -171.427, 95.729, 241.024]
  MoveL 836 to (-311.44, 0.85, 3.53) mm, rotated rx -179.15 ry 0 rz -30.08 deg; joints [8.851, -43.819, 139.84, -171.438, 95.763, 241.028]
  MoveL 837 to (-311.67, 0.44, 3.59) mm, rotated rx -179.15 ry 0 rz -30.08 deg; joints [8.839, -43.785, 139.837, -171.45, 95.794, 241.031]
  MoveL 838 to (-311.85, 0.14, 3.6) mm, rotated rx -179.15 ry 0 rz -30.08 deg; joints [8.829, -43.759, 139.833, -171.459, 95.816, 241.033]
  MoveL 839 to (-312.02, -0.16, 3.61) mm, rotated rx -179.15 ry 0 rz -30.08 deg; joints [8.82, -43.732, 139.827, -171.469, 95.837, 241.035]
  MoveL 840 to (-313.77, -3.18, 3.61) mm, rotated rx -179.15 ry 0 rz -30.08 deg; joints [8.724, -43.47, 139.772, -171.562, 96.043, 241.056]
  MoveL 841 to (-314.12, -3.78, 3.58) mm, rotated rx -179.15 ry 0 rz -30.08 deg; joints [8.705, -43.417, 139.759, -171.581, 96.083, 241.06]
  MoveL 842 to (-314.47, -4.39, 3.49) mm, rotated rx -179.15 ry 0 rz -30.08 deg; joints [8.685, -43.364, 139.741, -171.6, 96.118, 241.063]
  MoveL 843 to (-318.67, -11.63, 2.16) mm, rotated rx -179.15 ry 0 rz -30.08 deg; joints [8.443, -42.725, 139.509, -171.837, 96.525, 241.094]
  MoveL 844 to (-320.06, -14.04, 1.71) mm, rotated rx -179.15 ry 0 rz -30.08 deg; joints [8.363, -42.513, 139.43, -171.915, 96.658, 241.103]
  MoveL 845 to (-320.24, -14.34, 1.62) mm, rotated rx -179.15 ry 0 rz -30.08 deg; joints [8.353, -42.486, 139.418, -171.925, 96.672, 241.104]
  MoveL 846 to (-320.41, -14.63, 1.52) mm, rotated rx -179.15 ry 0 rz -30.08 deg; joints [8.342, -42.46, 139.404, -171.935, 96.685, 241.105]
  MoveL 847 to (-320.58, -14.93, 1.39) mm, rotated rx -179.15 ry 0 rz -30.08 deg; joints [8.332, -42.434, 139.389, -171.946, 96.696, 241.105]
  MoveL 848 to (-320.75, -15.22, 1.24) mm, rotated rx -179.15 ry 0 rz -30.08 deg; joints [8.321, -42.407, 139.373, -171.956, 96.707, 241.105]
  MoveL 849 to (-320.92, -15.52, 1.06) mm, rotated rx -179.15 ry 0 rz -30.08 deg; joints [8.31, -42.381, 139.354, -171.967, 96.715, 241.105]
  MoveL 850 to (-321.09, -15.82, 0.85) mm, rotated rx -179.15 ry 0 rz -30.08 deg; joints [8.299, -42.354, 139.334, -171.978, 96.722, 241.105]
  MoveL 851 to (-321.26, -16.11, 0.62) mm, rotated rx -179.15 ry 0 rz -30.08 deg; joints [8.288, -42.327, 139.312, -171.989, 96.726, 241.104]
  MoveL 852 to (-321.43, -16.41, 0.35) mm, rotated rx -179.15 ry 0 rz -30.08 deg; joints [8.276, -42.299, 139.287, -172.001, 96.729, 241.103]
  MoveL 853 to (-321.46, -16.46, 0.3) mm, rotated rx -179.15 ry 0 rz -30.08 deg; joints [8.274, -42.295, 139.282, -172.003, 96.729, 241.103]
  MoveC 854 to (-321.99, -17.38, 0.01) mm, rotated rx -179.15 ry 0 rz -30.08 deg; joints [8.243, -42.213, 139.244, -172.034, 96.772, 241.105] to (-322.44, -18.14, 0.66) mm, rotated rx -179.15 ry 0 rz -30.08 deg; joints [8.224, -42.151, 139.273, -172.052, 96.864, 241.115]
  MoveL 855 to (-322.44, -18.14, 0.66) mm, rotated rx -179.15 ry 0 rz -30.08 deg; joints [8.224, -42.151, 139.273, -172.052, 96.864, 241.115]
  MoveL 856 to (-323.43, -19.85, 4.32) mm, rotated rx -179.15 ry 0 rz -30.08 deg; joints [8.199, -42.023, 139.495, -172.071, 97.21, 241.161]
  MoveL 857 to (-324.83, -19.73, 5.44) mm, rotated rx -179.15 ry 0 rz -30.08 deg; joints [8.13, -42.039, 139.59, -172.139, 97.289, 241.163]
  Set speed (200.0 mm/s)
  MoveL 858 to (-336.31, -13.08, 5.44) mm, rotated rx -179.15 ry 0 rz -30.08 deg; joints [7.487, -42.624, 139.874, -172.792, 97.002, 241.04]
  Print: /'Parallel1'
  Call SetTool(1)
  Set speed (200.0 mm/s)
  MoveL 859 to (-340.11, 16.27, -316.36) mm, rotated rx -179.15 ry 0 rz -30.08 deg; joints [5.497, -38.983, 116.055, -174.698, 76.934, 238.948]
  MoveL 860 to (-319.42, 4.29, -316.36) mm, rotated rx -179.15 ry 0 rz -30.08 deg; joints [6.382, -38.16, 115.652, -173.801, 77.371, 238.793]
  Set speed (100.0 mm/s)
  MoveL 861 to (-318.78, 3.92, -316.36) mm, rotated rx -179.15 ry 0 rz -30.08 deg; joints [6.409, -38.135, 115.639, -173.773, 77.384, 238.788]
  MoveC 862 to (-318.01, 3.47, -315.99) mm, rotated rx -179.15 ry 0 rz -30.08 deg; joints [6.444, -38.114, 115.654, -173.738, 77.42, 238.784] to (-317.69, 3.28, -315.09) mm, rotated rx -179.15 ry 0 rz -30.08 deg; joints [6.462, -38.126, 115.721, -173.721, 77.476, 238.787]
  MoveL 863 to (-317.69, 3.28, -315.09) mm, rotated rx -179.15 ry 0 rz -30.08 deg; joints [6.462, -38.126, 115.721, -173.721, 77.476, 238.787]
  MoveL 864 to (-317.69, 3.28, 0.74) mm, rotated rx -179.15 ry 0 rz -30.08 deg; joints [8.481, -44.015, 139.77, -171.814, 95.505, 240.951]
  MoveL 865 to (-317.74, 3.32, 1.02) mm, rotated rx -179.15 ry 0 rz -30.08 deg; joints [8.48, -44.02, 139.791, -171.815, 95.521, 240.953]
  MoveL 866 to (-317.8, 3.35, 1.3) mm, rotated rx -179.15 ry 0 rz -30.08 deg; joints [8.479, -44.025, 139.812, -171.816, 95.537, 240.955]
  MoveL 867 to (-317.8, 3.35, 2.99) mm, rotated rx -179.15 ry 0 rz -30.08 deg; joints [8.493, -44.038, 139.931, -171.8, 95.642, 240.972]
  MoveC 868 to (-318.08, 2.86, 4.33) mm, rotated rx -179.15 ry 0 rz -30.08 deg; joints [8.489, -44.006, 140.017, -171.802, 95.758, 240.988] to (-318.75, 1.7, 4.89) mm, rotated rx -179.15 ry 0 rz -30.08 deg; joints [8.457, -43.909, 140.035, -171.833, 95.873, 241.001]
  MoveL 869 to (-318.75, 1.7, 4.89) mm, rotated rx -179.15 ry 0 rz -30.08 deg; joints [8.457, -43.909, 140.035, -171.833, 95.873, 241.001]
  MoveL 870 to (-320.03, -0.5, 4.89) mm, rotated rx -179.15 ry 0 rz -30.08 deg; joints [8.387, -43.717, 139.994, -171.901, 96.024, 241.015]
  MoveC 871 to (-320.7, -1.66, 4.33) mm, rotated rx -179.15 ry 0 rz -30.08 deg; joints [8.345, -43.611, 139.933, -171.943, 96.069, 241.017] to (-320.98, -2.15, 2.99) mm, rotated rx -179.15 ry 0 rz -30.08 deg; joints [8.318, -43.559, 139.829, -171.97, 96.018, 241.007]
  MoveL 872 to (-320.98, -2.15, 2.99) mm, rotated rx -179.15 ry 0 rz -30.08 deg; joints [8.318, -43.559, 139.829, -171.97, 96.018, 241.007]
  MoveL 873 to (-320.92, -2.18, 2.71) mm, rotated rx -179.15 ry 0 rz -30.08 deg; joints [8.319, -43.554, 139.808, -171.97, 96.002, 241.005]
  MoveL 874 to (-320.87, -2.21, 2.43) mm, rotated rx -179.15 ry 0 rz -30.08 deg; joints [8.32, -43.55, 139.787, -171.969, 95.986, 241.003]
  MoveL 875 to (-320.87, -2.21, -317.02) mm, rotated rx -179.15 ry 0 rz -30.08 deg; joints [6.318, -37.729, 115.484, -173.872, 77.632, 238.836]
  MoveL 876 to (-320.92, -2.18, -317.3) mm, rotated rx -179.15 ry 0 rz -30.08 deg; joints [6.315, -37.723, 115.462, -173.875, 77.616, 238.835]
  MoveL 877 to (-320.98, -2.15, -317.58) mm, rotated rx -179.15 ry 0 rz -30.08 deg; joints [6.311, -37.718, 115.44, -173.879, 77.599, 238.833]
  MoveL 878 to (-320.98, -2.15, -317.58) mm, rotated rx -179.15 ry 0 rz -30.08 deg; joints [6.311, -37.718, 115.44, -173.879, 77.599, 238.833]
  MoveC 879 to (-321.26, -2.63, -318.92) mm, rotated rx -179.15 ry 0 rz -30.08 deg; joints [6.293, -37.65, 115.322, -173.896, 77.548, 238.832] to (-321.94, -3.79, -319.48) mm, rotated rx -179.15 ry 0 rz -30.08 deg; joints [6.262, -37.562, 115.258, -173.928, 77.572, 238.841]
  MoveL 880 to (-321.94, -3.79, -319.48) mm, rotated rx -179.15 ry 0 rz -30.08 deg; joints [6.262, -37.562, 115.258, -173.928, 77.572, 238.841]
  MoveL 881 to (-323.21, -5.99, -319.48) mm, rotated rx -179.15 ry 0 rz -30.08 deg; joints [6.208, -37.425, 115.226, -173.986, 77.676, 238.864]
  MoveC 882 to (-323.88, -7.16, -318.92) mm, rotated rx -179.15 ry 0 rz -30.08 deg; joints [6.182, -37.367, 115.255, -174.014, 77.761, 238.879] to (-324.16, -7.64, -317.58) mm, rotated rx -179.15 ry 0 rz -30.08 deg; joints [6.177, -37.373, 115.359, -174.022, 77.859, 238.891]
  MoveL 883 to (-324.16, -7.64, -317.58) mm, rotated rx -179.15 ry 0 rz -30.08 deg; joints [6.177, -37.373, 115.359, -174.022, 77.859, 238.891]
  MoveL 884 to (-324.11, -7.67, -317.3) mm, rotated rx -179.15 ry 0 rz -30.08 deg; joints [6.18, -37.378, 115.381, -174.019, 77.875, 238.892]
  MoveL 885 to (-324.11, -7.67, -317.3) mm, rotated rx -179.15 ry 0 rz -30.08 deg; joints [6.181, -37.378, 115.381, -174.019, 77.875, 238.892]
  MoveL 886 to (-324.05, -7.7, -317.02) mm, rotated rx -179.15 ry 0 rz -30.08 deg; joints [6.184, -37.384, 115.403, -174.015, 77.892, 238.893]
  MoveL 887 to (-324.05, -7.7, 1.46) mm, rotated rx -179.15 ry 0 rz -30.08 deg; joints [8.137, -43.065, 139.615, -172.148, 96.298, 241.026]
  MoveC 888 to (-324.37, -7.52, 2.36) mm, rotated rx -179.15 ry 0 rz -30.08 deg; joints [8.127, -43.087, 139.685, -172.158, 96.346, 241.031] to (-325.15, -7.07, 2.73) mm, rotated rx -179.15 ry 0 rz -30.08 deg; joints [8.086, -43.129, 139.731, -172.199, 96.35, 241.027]
  MoveL 889 to (-325.15, -7.07, 2.73) mm, rotated rx -179.15 ry 0 rz -30.08 deg; joints [8.086, -43.129, 139.731, -172.199, 96.35, 241.027]
  Set speed (200.0 mm/s)
  MoveL 890 to (-346.48, 5.29, 2.73) mm, rotated rx -179.15 ry 0 rz -30.08 deg; joints [6.893, -44.221, 140.232, -173.406, 95.78, 240.822]
  MoveL 891 to (-346.48, 5.29, 2.73) mm, rotated rx -179.15 ry 0 rz -30.08 deg; joints [6.893, -44.221, 140.232, -173.406, 95.78, 240.822]

--- program Machining (robot KUKA KR 30 HA) ---
  Smooth(10)
  Print: /'1001'
  Print: /''
  Print: /'Contour3'
  Call SetTool(1)
  Set speed (200.0 mm/s)
  Set Ref.: Frame 3
  Set Tool: rc90 spindle mm
  Show rc90 spindle mm
  MoveJ 1 to (-334.45, 7.27, 4.38) mm, rotated rx -179.04 ry 0.05 rz -30.12 deg; joints [7.579, -44.36, 140.295, -172.73, 95.814, 240.847]
  MoveL 619 to (-335.6, -11.85, 4.35) mm, rotated rx -136.84 ry -38.16 rz -86.11 deg; joints [7.187, -50.278, 115.092, -236.827, 49.554, 234.918]
  MoveL 620 to (-332.9, -13.41, 4.35) mm, rotated rx -178.51 ry -54.99 rz -31.3 deg; joints [1.129, -38.512, 108.924, -239.668, 54.461, 270.428]
  Set speed (50.0 mm/s)
  MoveL 621 to (-326.98, -16.84, 4.35) mm, rotated rx -178.51 ry -54.99 rz -31.3 deg; joints [1.367, -38.307, 108.862, -239.327, 54.465, 270.227]
  MoveL 622 to (-325.36, -16.57, 3.64) mm, rotated rx -178.51 ry -54.99 rz -31.3 deg; joints [1.431, -38.297, 108.798, -239.291, 54.42, 270.27]
  Set speed (100.0 mm/s)
  MoveL 623 to (-324.39, -14.89, 2.31) mm, rotated rx -178.51 ry -54.99 rz -31.3 deg; joints [1.469, -38.349, 108.703, -239.342, 54.334, 270.418]
  MoveC 624 to (-324.11, -14.42, 1.33) mm, rotated rx -178.51 ry -54.99 rz -31.3 deg; joints [1.478, -38.343, 108.623, -239.377, 54.293, 270.494] to (-324.33, -14.8, 0.3) mm, rotated rx -178.51 ry -54.99 rz -31.3 deg; joints [1.469, -38.285, 108.526, -239.412, 54.276, 270.537]
  MoveL 625 to (-324.33, -14.8, 0.3) mm, rotated rx -178.51 ry -54.99 rz -31.3 deg; joints [1.469, -38.285, 108.526, -239.412, 54.276, 270.537]
  MoveL 626 to (-324.51, -15.11, -0.05) mm, rotated rx -178.51 ry -54.99 rz -31.3 deg; joints [1.461, -38.255, 108.492, -239.423, 54.276, 270.543]
  MoveL 627 to (-324.67, -15.38, -0.39) mm, rotated rx -178.51 ry -54.99 rz -31.3 deg; joints [1.454, -38.227, 108.458, -239.434, 54.275, 270.551]
  MoveL 628 to (-324.81, -15.61, -0.73) mm, rotated rx -178.51 ry -54.99 rz -31.3 deg; joints [1.449, -38.202, 108.424, -239.445, 54.273, 270.561]
  MoveL 629 to (-324.92, -15.82, -1.07) mm, rotated rx -178.51 ry -54.99 rz -31.3 deg; joints [1.444, -38.178, 108.391, -239.456, 54.269, 270.572]
  MoveL 630 to (-325.03, -15.99, -1.42) mm, rotated rx -178.51 ry -54.99 rz -31.3 deg; joints [1.439, -38.156, 108.358, -239.467, 54.265, 270.584]
  MoveL 631 to (-325.11, -16.15, -1.76) mm, rotated rx -178.51 ry -54.99 rz -31.3 deg; joints [1.435, -38.135, 108.326, -239.478, 54.261, 270.597]
  MoveL 632 to (-325.19, -16.28, -2.1) mm, rotated rx -178.51 ry -54.99 rz -31.3 deg; joints [1.432, -38.115, 108.294, -239.49, 54.255, 270.612]
  MoveL 633 to (-325.25, -16.39, -2.45) mm, rotated rx -178.51 ry -54.99 rz -31.3 deg; joints [1.429, -38.097, 108.262, -239.501, 54.249, 270.627]
  MoveL 634 to (-325.31, -16.48, -2.8) mm, rotated rx -178.51 ry -54.99 rz -31.3 deg; joints [1.427, -38.079, 108.229, -239.513, 54.242, 270.643]
  MoveL 635 to (-325.35, -16.55, -3.14) mm, rotated rx -178.51 ry -54.99 rz -31.3 deg; joints [1.424, -38.063, 108.197, -239.525, 54.235, 270.66]
  MoveL 636 to (-325.38, -16.61, -3.49) mm, rotated rx -178.51 ry -54.99 rz -31.3 deg; joints [1.423, -38.047, 108.166, -239.537, 54.227, 270.677]
  MoveL 637 to (-325.41, -16.65, -3.84) mm, rotated rx -178.51 ry -54.99 rz -31.3 deg; joints [1.422, -38.033, 108.134, -239.549, 54.219, 270.696]
  MoveL 638 to (-325.42, -16.67, -4.19) mm, rotated rx -178.51 ry -54.99 rz -31.3 deg; joints [1.421, -38.019, 108.103, -239.561, 54.21, 270.715]
  MoveL 639 to (-325.42, -16.68, -4.54) mm, rotated rx -178.51 ry -54.99 rz -31.3 deg; joints [1.42, -38.007, 108.071, -239.573, 54.201, 270.735]
  MoveL 640 to (-325.42, -16.68, -311.19) mm, rotated rx -178.51 ry -54.99 rz -31.3 deg; joints [1.154, -24.591, 76.575, -253.619, 47.036, 292.306]
  MoveL 641 to (-325.42, -16.67, -311.54) mm, rotated rx -178.51 ry -54.99 rz -31.3 deg; joints [1.154, -24.572, 76.532, -253.641, 47.03, 292.337]
  MoveL 642 to (-325.41, -16.65, -311.88) mm, rotated rx -178.51 ry -54.99 rz -31.3 deg; joints [1.154, -24.553, 76.49, -253.662, 47.023, 292.369]
  MoveL 643 to (-325.38, -16.61, -312.23) mm, rotated rx -178.51 ry -54.99 rz -31.3 deg; joints [1.154, -24.536, 76.447, -253.684, 47.015, 292.402]
  MoveL 644 to (-325.35, -16.55, -312.58) mm, rotated rx -178.51 ry -54.99 rz -31.3 deg; joints [1.155, -24.519, 76.405, -253.706, 47.008, 292.435]
  MoveL 645 to (-325.31, -16.48, -312.93) mm, rotated rx -178.51 ry -54.99 rz -31.3 deg; joints [1.156, -24.503, 76.363, -253.729, 47, 292.469]
  MoveL 646 to (-325.25, -16.39, -313.28) mm, rotated rx -178.51 ry -54.99 rz -31.3 deg; joints [1.158, -24.488, 76.321, -253.751, 46.991, 292.504]
  MoveL 647 to (-325.19, -16.27, -313.63) mm, rotated rx -178.51 ry -54.99 rz -31.3 deg; joints [1.16, -24.474, 76.28, -253.774, 46.983, 292.54]
  MoveL 648 to (-325.11, -16.14, -313.98) mm, rotated rx -178.51 ry -54.99 rz -31.3 deg; joints [1.162, -24.461, 76.238, -253.797, 46.973, 292.576]
  MoveL 649 to (-325.02, -15.98, -314.33) mm, rotated rx -178.51 ry -54.99 rz -31.3 deg; joints [1.165, -24.449, 76.197, -253.82, 46.964, 292.614]
  MoveL 650 to (-324.91, -15.8, -314.68) mm, rotated rx -178.51 ry -54.99 rz -31.3 deg; joints [1.168, -24.438, 76.157, -253.844, 46.953, 292.652]
  MoveL 651 to (-324.79, -15.59, -315.03) mm, rotated rx -178.51 ry -54.99 rz -31.3 deg; joints [1.172, -24.429, 76.117, -253.868, 46.943, 292.691]
  MoveL 652 to (-324.65, -15.35, -315.38) mm, rotated rx -178.51 ry -54.99 rz -31.3 deg; joints [1.176, -24.421, 76.077, -253.893, 46.931, 292.732]
  MoveL 653 to (-324.5, -15.09, -315.7) mm, rotated rx -178.51 ry -54.99 rz -31.3 deg; joints [1.181, -24.415, 76.041, -253.915, 46.92, 292.771]
  MoveL 654 to (-324.33, -14.8, -316.02) mm, rotated rx -178.51 ry -54.99 rz -31.3 deg; joints [1.186, -24.411, 76.005, -253.939, 46.908, 292.812]
  MoveL 655 to (-324.16, -14.49, -316.3) mm, rotated rx -178.51 ry -54.99 rz -31.3 deg; joints [1.191, -24.409, 75.974, -253.96, 46.897, 292.849]
  MoveL 656 to (-323.98, -14.19, -316.55) mm, rotated rx -178.51 ry -54.99 rz -31.3 deg; joints [1.197, -24.41, 75.948, -253.979, 46.886, 292.883]
  MoveL 657 to (-323.81, -13.89, -316.76) mm, rotated rx -178.51 ry -54.99 rz -31.3 deg; joints [1.203, -24.412, 75.926, -253.996, 46.876, 292.914]
  MoveL 658 to (-323.63, -13.59, -316.95) mm, rotated rx -178.51 ry -54.99 rz -31.3 deg; joints [1.208, -24.416, 75.907, -254.011, 46.867, 292.942]
  MoveL 659 to (-323.46, -13.29, -317.1) mm, rotated rx -178.51 ry -54.99 rz -31.3 deg; joints [1.214, -24.422, 75.892, -254.024, 46.857, 292.968]
  MoveL 660 to (-323.28, -12.99, -317.23) mm, rotated rx -178.51 ry -54.99 rz -31.3 deg; joints [1.219, -24.429, 75.88, -254.036, 46.849, 292.992]
  MoveL 661 to (-323.11, -12.68, -317.34) mm, rotated rx -178.51 ry -54.99 rz -31.3 deg; joints [1.225, -24.437, 75.87, -254.047, 46.841, 293.014]
  MoveL 662 to (-322.93, -12.38, -317.43) mm, rotated rx -178.51 ry -54.99 rz -31.3 deg; joints [1.23, -24.446, 75.864, -254.056, 46.833, 293.034]
  MoveL 663 to (-322.76, -12.08, -317.5) mm, rotated rx -178.51 ry -54.99 rz -31.3 deg; joints [1.236, -24.456, 75.86, -254.064, 46.826, 293.052]
  MoveL 664 to (-322.58, -11.78, -317.55) mm, rotated rx -178.51 ry -54.99 rz -31.3 deg; joints [1.242, -24.468, 75.858, -254.07, 46.818, 293.068]
  MoveL 665 to (-322.41, -11.48, -317.58) mm, rotated rx -178.51 ry -54.99 rz -31.3 deg; joints [1.247, -24.481, 75.858, -254.076, 46.812, 293.082]
  MoveL 666 to (-322.23, -11.17, -317.59) mm, rotated rx -178.51 ry -54.99 rz -31.3 deg; joints [1.253, -24.495, 75.862, -254.08, 46.805, 293.095]
  MoveL 667 to (-315.94, -0.31, -317.59) mm, rotated rx -178.51 ry -54.99 rz -31.3 deg; joints [1.458, -25.005, 76.005, -254.22, 46.582, 293.531]
  MoveL 668 to (-315.59, 0.29, -317.58) mm, rotated rx -178.51 ry -54.99 rz -31.3 deg; joints [1.469, -25.034, 76.014, -254.227, 46.57, 293.555]
  MoveL 669 to (-315.42, 0.6, -317.55) mm, rotated rx -178.51 ry -54.99 rz -31.3 deg; joints [1.475, -25.049, 76.022, -254.23, 46.564, 293.565]
  MoveL 670 to (-315.24, 0.9, -317.5) mm, rotated rx -178.51 ry -54.99 rz -31.3 deg; joints [1.481, -25.066, 76.031, -254.231, 46.559, 293.573]
  MoveL 671 to (-315.07, 1.2, -317.43) mm, rotated rx -178.51 ry -54.99 rz -31.3 deg; joints [1.486, -25.084, 76.043, -254.231, 46.553, 293.579]
  MoveL 672 to (-314.89, 1.5, -317.34) mm, rotated rx -178.51 ry -54.99 rz -31.3 deg; joints [1.492, -25.103, 76.058, -254.229, 46.549, 293.583]
  MoveL 673 to (-314.72, 1.8, -317.23) mm, rotated rx -178.51 ry -54.99 rz -31.3 deg; joints [1.498, -25.123, 76.076, -254.226, 46.545, 293.586]
  MoveL 674 to (-314.54, 2.1, -317.1) mm, rotated rx -178.51 ry -54.99 rz -31.3 deg; joints [1.504, -25.145, 76.096, -254.222, 46.541, 293.586]
  MoveL 675 to (-314.39, 2.36, -316.97) mm, rotated rx -178.51 ry -54.99 rz -31.3 deg; joints [1.509, -25.164, 76.115, -254.217, 46.538, 293.585]
  MoveL 676 to (-314.24, 2.62, -316.82) mm, rotated rx -178.51 ry -54.99 rz -31.3 deg; joints [1.514, -25.185, 76.137, -254.211, 46.535, 293.582]
  MoveL 677 to (-314.09, 2.88, -316.65) mm, rotated rx -178.51 ry -54.99 rz -31.3 deg; joints [1.519, -25.207, 76.162, -254.204, 46.533, 293.577]
  MoveL 678 to (-313.95, 3.13, -316.45) mm, rotated rx -178.51 ry -54.99 rz -31.3 deg; joints [1.524, -25.23, 76.189, -254.196, 46.531, 293.57]
  MoveL 679 to (-313.8, 3.39, -316.23) mm, rotated rx -178.51 ry -54.99 rz -31.3 deg; joints [1.529, -25.254, 76.219, -254.185, 46.529, 293.561]
  MoveL 680 to (-313.65, 3.65, -315.98) mm, rotated rx -178.51 ry -54.99 rz -31.3 deg; joints [1.534, -25.28, 76.253, -254.173, 46.528, 293.549]
  MoveL 681 to (-313.49, 3.92, -315.68) mm, rotated rx -178.51 ry -54.99 rz -31.3 deg; joints [1.539, -25.31, 76.294, -254.158, 46.528, 293.534]
  MoveL 682 to (-313.35, 4.16, -315.38) mm, rotated rx -178.51 ry -54.99 rz -31.3 deg; joints [1.544, -25.338, 76.334, -254.143, 46.529, 293.516]
  MoveL 683 to (-313.24, 4.35, -315.11) mm, rotated rx -178.51 ry -54.99 rz -31.3 deg; joints [1.548, -25.362, 76.369, -254.129, 46.529, 293.5]
  MoveL 684 to (-313.14, 4.52, -314.85) mm, rotated rx -178.51 ry -54.99 rz -31.3 deg; joints [1.551, -25.384, 76.404, -254.115, 46.531, 293.484]
  MoveL 685 to (-313.05, 4.68, -314.57) mm, rotated rx -178.51 ry -54.99 rz -31.3 deg; joints [1.555, -25.408, 76.441, -254.099, 46.532, 293.465]
  MoveL 686 to (-312.97, 4.82, -314.28) mm, rotated rx -178.51 ry -54.99 rz -31.3 deg; joints [1.557, -25.43, 76.478, -254.084, 46.534, 293.446]
  MoveL 687 to (-312.9, 4.95, -314) mm, rotated rx -178.51 ry -54.99 rz -31.3 deg; joints [1.56, -25.452, 76.514, -254.068, 46.537, 293.425]
  MoveL 688 to (-312.83, 5.06, -313.72) mm, rotated rx -178.51 ry -54.99 rz -31.3 deg; joints [1.563, -25.473, 76.55, -254.052, 46.54, 293.405]
  MoveL 689 to (-312.73, 5.24, -313.15) mm, rotated rx -178.51 ry -54.99 rz -31.3 deg; joints [1.566, -25.513, 76.622, -254.019, 46.546, 293.362]
  MoveL 690 to (-312.65, 5.37, -312.58) mm, rotated rx -178.51 ry -54.99 rz -31.3 deg; joints [1.569, -25.551, 76.694, -253.986, 46.553, 293.317]
  MoveL 691 to (-312.62, 5.43, -312.23) mm, rotated rx -178.51 ry -54.99 rz -31.3 deg; joints [1.571, -25.573, 76.737, -253.965, 46.558, 293.288]
  MoveL 692 to (-312.59, 5.47, -311.88) mm, rotated rx -178.51 ry -54.99 rz -31.3 deg; joints [1.572, -25.595, 76.781, -253.944, 46.564, 293.259]
  MoveL 693 to (-312.58, 5.49, -311.54) mm, rotated rx -178.51 ry -54.99 rz -31.3 deg; joints [1.573, -25.615, 76.824, -253.922, 46.57, 293.229]
  MoveL 694 to (-312.58, 5.49, -311.19) mm, rotated rx -178.51 ry -54.99 rz -31.3 deg; joints [1.573, -25.635, 76.867, -253.901, 46.576, 293.198]
  MoveL 695 to (-312.58, 5.49, -5.24) mm, rotated rx -178.51 ry -54.99 rz -31.3 deg; joints [1.928, -39.26, 108.282, -239.689, 53.521, 271.738]
  MoveL 696 to (-312.58, 5.49, -2.45) mm, rotated rx -178.51 ry -54.99 rz -31.3 deg; joints [1.931, -39.36, 108.53, -239.59, 53.595, 271.578]
  MoveL 697 to (-312.59, 5.47, -2.1) mm, rotated rx -178.51 ry -54.99 rz -31.3 deg; joints [1.931, -39.371, 108.561, -239.578, 53.605, 271.557]
  MoveL 698 to (-312.62, 5.43, -1.75) mm, rotated rx -178.51 ry -54.99 rz -31.3 deg; joints [1.931, -39.381, 108.592, -239.565, 53.615, 271.535]
  MoveL 699 to (-312.65, 5.37, -1.4) mm, rotated rx -178.51 ry -54.99 rz -31.3 deg; joints [1.93, -39.391, 108.622, -239.553, 53.626, 271.512]
  MoveL 700 to (-312.69, 5.3, -1.05) mm, rotated rx -178.51 ry -54.99 rz -31.3 deg; joints [1.929, -39.399, 108.652, -239.54, 53.637, 271.489]
  MoveL 701 to (-312.75, 5.2, -0.7) mm, rotated rx -178.51 ry -54.99 rz -31.3 deg; joints [1.927, -39.406, 108.682, -239.527, 53.65, 271.465]
  MoveL 702 to (-312.81, 5.09, -0.35) mm, rotated rx -178.51 ry -54.99 rz -31.3 deg; joints [1.925, -39.412, 108.712, -239.515, 53.662, 271.44]
  MoveL 703 to (-312.89, 4.96, 0) mm, rotated rx -178.51 ry -54.99 rz -31.3 deg; joints [1.923, -39.417, 108.742, -239.502, 53.676, 271.414]
  MoveL 704 to (-312.98, 4.8, 0.35) mm, rotated rx -178.51 ry -54.99 rz -31.3 deg; joints [1.92, -39.42, 108.771, -239.489, 53.69, 271.388]
  MoveL 705 to (-313.06, 4.67, 0.61) mm, rotated rx -178.51 ry -54.99 rz -31.3 deg; joints [1.917, -39.422, 108.793, -239.479, 53.7, 271.367]
  MoveL 706 to (-313.14, 4.52, 0.87) mm, rotated rx -178.51 ry -54.99 rz -31.3 deg; joints [1.914, -39.423, 108.814, -239.469, 53.712, 271.345]
  MoveL 707 to (-313.28, 4.28, 1.23) mm, rotated rx -178.51 ry -54.99 rz -31.3 deg; joints [1.909, -39.422, 108.844, -239.455, 53.729, 271.314]
  MoveL 708 to (-313.44, 4.01, 1.6) mm, rotated rx -178.51 ry -54.99 rz -31.3 deg; joints [1.903, -39.419, 108.873, -239.441, 53.747, 271.281]
  MoveL 709 to (-313.54, 3.84, 1.8) mm, rotated rx -178.51 ry -54.99 rz -31.3 deg; joints [1.899, -39.417, 108.889, -239.433, 53.757, 271.262]
  MoveL 710 to (-313.64, 3.66, 1.99) mm, rotated rx -178.51 ry -54.99 rz -31.3 deg; joints [1.896, -39.413, 108.904, -239.426, 53.768, 271.244]
  MoveL 711 to (-313.84, 3.31, 2.32) mm, rotated rx -178.51 ry -54.99 rz -31.3 deg; joints [1.888, -39.405, 108.929, -239.413, 53.787, 271.209]
  MoveL 712 to (-314.02, 3.01, 2.57) mm, rotated rx -178.51 ry -54.99 rz -31.3 deg; joints [1.881, -39.396, 108.948, -239.403, 53.803, 271.182]
  MoveL 713 to (-314.19, 2.71, 2.78) mm, rotated rx -178.51 ry -54.99 rz -31.3 deg; joints [1.875, -39.386, 108.963, -239.394, 53.818, 271.156]
  MoveL 714 to (-314.37, 2.41, 2.96) mm, rotated rx -178.51 ry -54.99 rz -31.3 deg; joints [1.868, -39.376, 108.976, -239.386, 53.832, 271.133]
  MoveL 715 to (-314.54, 2.1, 3.12) mm, rotated rx -178.51 ry -54.99 rz -31.3 deg; joints [1.861, -39.364, 108.986, -239.379, 53.845, 271.11]
  MoveL 716 to (-314.57, 2.06, 3.14) mm, rotated rx -178.51 ry -54.99 rz -31.3 deg; joints [1.86, -39.362, 108.987, -239.378, 53.847, 271.107]
  MoveL 717 to (-314.74, 1.76, 3.27) mm, rotated rx -178.51 ry -54.99 rz -31.3 deg; joints [1.854, -39.349, 108.995, -239.373, 53.86, 271.087]
  MoveL 718 to (-314.91, 1.47, 3.37) mm, rotated rx -178.51 ry -54.99 rz -31.3 deg; joints [1.847, -39.336, 109.001, -239.368, 53.871, 271.068]
  MoveL 719 to (-315.08, 1.17, 3.46) mm, rotated rx -178.51 ry -54.99 rz -31.3 deg; joints [1.84, -39.322, 109.005, -239.364, 53.883, 271.05]
  MoveL 720 to (-315.25, 0.88, 3.52) mm, rotated rx -178.51 ry -54.99 rz -31.3 deg; joints [1.834, -39.307, 109.008, -239.36, 53.893, 271.033]
  MoveL 721 to (-315.43, 0.58, 3.57) mm, rotated rx -178.51 ry -54.99 rz -31.3 deg; joints [1.827, -39.292, 109.008, -239.357, 53.904, 271.018]
  MoveL 722 to (-315.6, 0.28, 3.6) mm, rotated rx -178.51 ry -54.99 rz -31.3 deg; joints [1.82, -39.275, 109.007, -239.355, 53.913, 271.003]
  MoveL 723 to (-315.94, -0.31, 3.61) mm, rotated rx -178.51 ry -54.99 rz -31.3 deg; joints [1.806, -39.241, 109.001, -239.352, 53.932, 270.976]
  MoveL 724 to (-316.64, -1.52, 3.61) mm, rotated rx -178.51 ry -54.99 rz -31.3 deg; joints [1.779, -39.171, 108.987, -239.347, 53.968, 270.923]
  MoveL 725 to (-316.99, -2.12, 3.58) mm, rotated rx -178.51 ry -54.99 rz -31.3 deg; joints [1.765, -39.136, 108.977, -239.345, 53.986, 270.898]
  MoveL 726 to (-317.34, -2.72, 3.49) mm, rotated rx -178.51 ry -54.99 rz -31.3 deg; joints [1.751, -39.098, 108.962, -239.346, 54.002, 270.877]
  MoveL 727 to (-321.53, -9.97, 2.16) mm, rotated rx -178.51 ry -54.99 rz -31.3 deg; joints [1.582, -38.631, 108.755, -239.364, 54.183, 270.638]
  MoveL 728 to (-322.93, -12.38, 1.71) mm, rotated rx -178.51 ry -54.99 rz -31.3 deg; joints [1.526, -38.475, 108.683, -239.371, 54.243, 270.56]
  MoveL 729 to (-323.1, -12.68, 1.62) mm, rotated rx -178.51 ry -54.99 rz -31.3 deg; joints [1.519, -38.454, 108.672, -239.373, 54.25, 270.552]
  MoveL 730 to (-323.28, -12.97, 1.52) mm, rotated rx -178.51 ry -54.99 rz -31.3 deg; joints [1.512, -38.433, 108.658, -239.376, 54.255, 270.545]
  MoveL 731 to (-323.45, -13.27, 1.39) mm, rotated rx -178.51 ry -54.99 rz -31.3 deg; joints [1.505, -38.412, 108.643, -239.379, 54.261, 270.54]
  MoveL 732 to (-323.62, -13.56, 1.24) mm, rotated rx -178.51 ry -54.99 rz -31.3 deg; joints [1.498, -38.389, 108.626, -239.384, 54.265, 270.536]
  MoveL 733 to (-323.79, -13.86, 1.06) mm, rotated rx -178.51 ry -54.99 rz -31.3 deg; joints [1.491, -38.366, 108.606, -239.389, 54.269, 270.533]
  MoveL 734 to (-323.96, -14.15, 0.85) mm, rotated rx -178.51 ry -54.99 rz -31.3 deg; joints [1.484, -38.342, 108.584, -239.395, 54.273, 270.532]
  MoveL 735 to (-324.13, -14.45, 0.62) mm, rotated rx -178.51 ry -54.99 rz -31.3 deg; joints [1.477, -38.316, 108.559, -239.402, 54.275, 270.533]
  MoveL 736 to (-324.3, -14.75, 0.35) mm, rotated rx -178.51 ry -54.99 rz -31.3 deg; joints [1.47, -38.29, 108.532, -239.41, 54.276, 270.536]
  MoveL 737 to (-324.33, -14.8, 0.3) mm, rotated rx -178.51 ry -54.99 rz -31.3 deg; joints [1.469, -38.285, 108.526, -239.412, 54.276, 270.537]
  MoveC 738 to (-325.22, -16.33, 0.41) mm, rotated rx -178.51 ry -54.99 rz -31.3 deg; joints [1.433, -38.2, 108.516, -239.403, 54.325, 270.465] to (-325.18, -16.27, 2.18) mm, rotated rx -178.51 ry -54.99 rz -31.3 deg; joints [1.437, -38.265, 108.674, -239.342, 54.371, 270.366]
  MoveL 739 to (-325.18, -16.27, 2.18) mm, rotated rx -178.51 ry -54.99 rz -31.3 deg; joints [1.437, -38.265, 108.674, -239.342, 54.371, 270.366]
  MoveL 740 to (-324.74, -15.51, 3.02) mm, rotated rx -178.51 ry -54.99 rz -31.3 deg; joints [1.455, -38.338, 108.758, -239.316, 54.371, 270.351]
  Set speed (50.0 mm/s)
  MoveL 741 to (-322.97, -16.53, 3.02) mm, rotated rx -178.51 ry -54.99 rz -31.3 deg; joints [1.526, -38.277, 108.739, -239.214, 54.372, 270.291]
  MoveL 742 to (-321.44, -16.41, 2.09) mm, rotated rx -178.51 ry -54.99 rz -31.3 deg; joints [1.587, -38.25, 108.655, -239.185, 54.325, 270.339]
  Set speed (100.0 mm/s)
  MoveC 743 to (-321.26, -16.11, 1.18) mm, rotated rx -178.51 ry -54.99 rz -31.3 deg; joints [1.593, -38.236, 108.578, -239.218, 54.292, 270.404] to (-321.46, -16.46, 0.3) mm, rotated rx -178.51 ry -54.99 rz -31.3 deg; joints [1.584, -38.185, 108.495, -239.247, 54.278, 270.44]
  MoveL 744 to (-321.46, -16.46, 0.3) mm, rotated rx -178.51 ry -54.99 rz -31.3 deg; joints [1.584, -38.185, 108.495, -239.247, 54.278, 270.44]
  MoveL 745 to (-321.65, -16.77, -0.05) mm, rotated rx -178.51 ry -54.99 rz -31.3 deg; joints [1.576, -38.155, 108.46, -239.258, 54.278, 270.447]
  MoveL 746 to (-321.8, -17.04, -0.39) mm, rotated rx -178.51 ry -54.99 rz -31.3 deg; joints [1.569, -38.128, 108.426, -239.269, 54.276, 270.455]
  MoveL 747 to (-321.94, -17.28, -0.73) mm, rotated rx -178.51 ry -54.99 rz -31.3 deg; joints [1.564, -38.102, 108.393, -239.28, 54.274, 270.465]
  MoveL 748 to (-322.05, -17.48, -1.07) mm, rotated rx -178.51 ry -54.99 rz -31.3 deg; joints [1.559, -38.078, 108.36, -239.291, 54.271, 270.476]
  MoveL 749 to (-322.16, -17.66, -1.42) mm, rotated rx -178.51 ry -54.99 rz -31.3 deg; joints [1.554, -38.056, 108.327, -239.303, 54.267, 270.488]
  MoveL 750 to (-322.25, -17.81, -1.76) mm, rotated rx -178.51 ry -54.99 rz -31.3 deg; joints [1.55, -38.035, 108.294, -239.314, 54.262, 270.501]
  MoveL 751 to (-322.32, -17.94, -2.1) mm, rotated rx -178.51 ry -54.99 rz -31.3 deg; joints [1.547, -38.016, 108.262, -239.325, 54.256, 270.515]
  MoveL 752 to (-322.38, -18.05, -2.45) mm, rotated rx -178.51 ry -54.99 rz -31.3 deg; joints [1.544, -37.998, 108.23, -239.337, 54.25, 270.53]
  MoveL 753 to (-322.44, -18.14, -2.8) mm, rotated rx -178.51 ry -54.99 rz -31.3 deg; joints [1.541, -37.98, 108.198, -239.349, 54.243, 270.546]
  MoveL 754 to (-322.48, -18.22, -3.14) mm, rotated rx -178.51 ry -54.99 rz -31.3 deg; joints [1.539, -37.964, 108.166, -239.361, 54.236, 270.563]
  MoveL 755 to (-322.51, -18.27, -3.49) mm, rotated rx -178.51 ry -54.99 rz -31.3 deg; joints [1.538, -37.948, 108.134, -239.373, 54.228, 270.581]
  MoveL 756 to (-322.54, -18.31, -3.84) mm, rotated rx -178.51 ry -54.99 rz -31.3 deg; joints [1.536, -37.934, 108.103, -239.385, 54.22, 270.6]
  MoveL 757 to (-322.55, -18.34, -4.19) mm, rotated rx -178.51 ry -54.99 rz -31.3 deg; joints [1.535, -37.92, 108.071, -239.397, 54.211, 270.619]
  MoveL 758 to (-322.55, -18.34, -4.54) mm, rotated rx -178.51 ry -54.99 rz -31.3 deg; joints [1.535, -37.908, 108.04, -239.409, 54.202, 270.639]
  MoveL 759 to (-322.55, -18.34, -311.19) mm, rotated rx -178.51 ry -54.99 rz -31.3 deg; joints [1.248, -24.507, 76.541, -253.486, 46.994, 292.219]
  MoveL 760 to (-322.55, -18.33, -311.54) mm, rotated rx -178.51 ry -54.99 rz -31.3 deg; joints [1.248, -24.488, 76.498, -253.507, 46.988, 292.251]
  MoveL 761 to (-322.54, -18.31, -311.88) mm, rotated rx -178.51 ry -54.99 rz -31.3 deg; joints [1.248, -24.47, 76.455, -253.529, 46.981, 292.283]
  MoveL 762 to (-322.51, -18.27, -312.23) mm, rotated rx -178.51 ry -54.99 rz -31.3 deg; joints [1.249, -24.453, 76.413, -253.551, 46.973, 292.315]
  MoveL 763 to (-322.48, -18.22, -312.58) mm, rotated rx -178.51 ry -54.99 rz -31.3 deg; joints [1.25, -24.436, 76.371, -253.573, 46.966, 292.349]
  MoveL 764 to (-322.44, -18.14, -312.93) mm, rotated rx -178.51 ry -54.99 rz -31.3 deg; joints [1.251, -24.42, 76.329, -253.595, 46.958, 292.383]
  MoveL 765 to (-322.38, -18.05, -313.28) mm, rotated rx -178.51 ry -54.99 rz -31.3 deg; joints [1.252, -24.405, 76.287, -253.618, 46.949, 292.418]
  MoveL 766 to (-322.32, -17.93, -313.63) mm, rotated rx -178.51 ry -54.99 rz -31.3 deg; joints [1.254, -24.391, 76.245, -253.641, 46.94, 292.453]
  MoveL 767 to (-322.24, -17.8, -313.98) mm, rotated rx -178.51 ry -54.99 rz -31.3 deg; joints [1.257, -24.378, 76.204, -253.664, 46.931, 292.49]
  MoveL 768 to (-322.15, -17.64, -314.33) mm, rotated rx -178.51 ry -54.99 rz -31.3 deg; joints [1.259, -24.366, 76.163, -253.687, 46.921, 292.527]
  MoveL 769 to (-322.05, -17.46, -314.68) mm, rotated rx -178.51 ry -54.99 rz -31.3 deg; joints [1.262, -24.355, 76.122, -253.711, 46.911, 292.566]
  MoveL 770 to (-321.92, -17.25, -315.03) mm, rotated rx -178.51 ry -54.99 rz -31.3 deg; joints [1.266, -24.345, 76.082, -253.735, 46.9, 292.605]
  MoveL 771 to (-321.78, -17.01, -315.38) mm, rotated rx -178.51 ry -54.99 rz -31.3 deg; joints [1.27, -24.337, 76.042, -253.76, 46.889, 292.646]
  MoveL 772 to (-321.63, -16.75, -315.7) mm, rotated rx -178.51 ry -54.99 rz -31.3 deg; joints [1.275, -24.332, 76.006, -253.783, 46.877, 292.685]
  MoveL 773 to (-321.46, -16.46, -316.02) mm, rotated rx -178.51 ry -54.99 rz -31.3 deg; joints [1.28, -24.328, 75.97, -253.806, 46.865, 292.725]
  MoveL 774 to (-321.29, -16.16, -316.3) mm, rotated rx -178.51 ry -54.99 rz -31.3 deg; joints [1.286, -24.326, 75.94, -253.827, 46.854, 292.763]
  MoveL 775 to (-321.11, -15.85, -316.55) mm, rotated rx -178.51 ry -54.99 rz -31.3 deg; joints [1.291, -24.327, 75.913, -253.846, 46.843, 292.797]
  MoveL 776 to (-320.94, -15.55, -316.76) mm, rotated rx -178.51 ry -54.99 rz -31.3 deg; joints [1.297, -24.329, 75.891, -253.863, 46.833, 292.827]
  MoveL 777 to (-320.76, -15.25, -316.94) mm, rotated rx -178.51 ry -54.99 rz -31.3 deg; joints [1.302, -24.333, 75.873, -253.878, 46.824, 292.856]
  MoveL 778 to (-320.59, -14.95, -317.1) mm, rotated rx -178.51 ry -54.99 rz -31.3 deg; joints [1.308, -24.339, 75.858, -253.892, 46.815, 292.882]
  MoveL 779 to (-320.41, -14.65, -317.23) mm, rotated rx -178.51 ry -54.99 rz -31.3 deg; joints [1.313, -24.346, 75.845, -253.903, 46.806, 292.906]
  MoveL 780 to (-320.24, -14.35, -317.34) mm, rotated rx -178.51 ry -54.99 rz -31.3 deg; joints [1.319, -24.354, 75.836, -253.914, 46.798, 292.927]
  MoveL 781 to (-320.06, -14.04, -317.43) mm, rotated rx -178.51 ry -54.99 rz -31.3 deg; joints [1.325, -24.363, 75.829, -253.923, 46.79, 292.947]
  MoveL 782 to (-319.89, -13.74, -317.5) mm, rotated rx -178.51 ry -54.99 rz -31.3 deg; joints [1.33, -24.373, 75.825, -253.931, 46.782, 292.965]
  MoveL 783 to (-319.71, -13.44, -317.55) mm, rotated rx -178.51 ry -54.99 rz -31.3 deg; joints [1.336, -24.385, 75.823, -253.938, 46.775, 292.981]
  MoveL 784 to (-319.54, -13.14, -317.58) mm, rotated rx -178.51 ry -54.99 rz -31.3 deg; joints [1.342, -24.398, 75.824, -253.943, 46.769, 292.996]
  MoveL 785 to (-319.37, -12.84, -317.59) mm, rotated rx -178.51 ry -54.99 rz -31.3 deg; joints [1.347, -24.412, 75.827, -253.948, 46.762, 293.009]
  MoveL 786 to (-312.02, -0.16, -317.59) mm, rotated rx -178.51 ry -54.99 rz -31.3 deg; joints [1.586, -25.006, 75.994, -254.111, 46.501, 293.518]
  MoveL 787 to (-311.85, 0.14, -317.58) mm, rotated rx -178.51 ry -54.99 rz -31.3 deg; joints [1.592, -25.021, 75.998, -254.115, 46.495, 293.53]
  MoveL 788 to (-311.67, 0.44, -317.56) mm, rotated rx -178.51 ry -54.99 rz -31.3 deg; joints [1.597, -25.036, 76.004, -254.118, 46.489, 293.541]
  MoveL 789 to (-311.5, 0.74, -317.53) mm, rotated rx -178.51 ry -54.99 rz -31.3 deg; joints [1.603, -25.052, 76.013, -254.12, 46.483, 293.55]
  MoveL 790 to (-311.32, 1.05, -317.47) mm, rotated rx -178.51 ry -54.99 rz -31.3 deg; joints [1.609, -25.069, 76.024, -254.12, 46.478, 293.557]
  MoveL 791 to (-311.15, 1.35, -317.39) mm, rotated rx -178.51 ry -54.99 rz -31.3 deg; joints [1.615, -25.088, 76.037, -254.119, 46.473, 293.562]
  MoveL 792 to (-310.97, 1.65, -317.29) mm, rotated rx -178.51 ry -54.99 rz -31.3 deg; joints [1.62, -25.107, 76.053, -254.117, 46.468, 293.566]
  MoveL 793 to (-310.8, 1.95, -317.17) mm, rotated rx -178.51 ry -54.99 rz -31.3 deg; joints [1.626, -25.128, 76.072, -254.114, 46.464, 293.567]
  MoveL 794 to (-310.62, 2.25, -317.03) mm, rotated rx -178.51 ry -54.99 rz -31.3 deg; joints [1.632, -25.15, 76.093, -254.109, 46.461, 293.567]
  MoveL 795 to (-310.45, 2.55, -316.86) mm, rotated rx -178.51 ry -54.99 rz -31.3 deg; joints [1.638, -25.174, 76.118, -254.102, 46.457, 293.564]
  MoveL 796 to (-310.28, 2.86, -316.66) mm, rotated rx -178.51 ry -54.99 rz -31.3 deg; joints [1.644, -25.199, 76.146, -254.094, 46.455, 293.558]
  MoveL 797 to (-310.09, 3.18, -316.41) mm, rotated rx -178.51 ry -54.99 rz -31.3 deg; joints [1.65, -25.229, 76.181, -254.083, 46.452, 293.55]
  MoveL 798 to (-309.9, 3.51, -316.12) mm, rotated rx -178.51 ry -54.99 rz -31.3 deg; joints [1.657, -25.26, 76.221, -254.069, 46.451, 293.537]
  MoveL 799 to (-309.71, 3.84, -315.78) mm, rotated rx -178.51 ry -54.99 rz -31.3 deg; joints [1.663, -25.295, 76.267, -254.053, 46.45, 293.52]
  MoveL 800 to (-309.52, 4.16, -315.38) mm, rotated rx -178.51 ry -54.99 rz -31.3 deg; joints [1.67, -25.332, 76.321, -254.032, 46.45, 293.497]
  MoveL 801 to (-309.4, 4.37, -315.08) mm, rotated rx -178.51 ry -54.99 rz -31.3 deg; joints [1.674, -25.359, 76.359, -254.016, 46.451, 293.48]
  MoveL 802 to (-309.29, 4.55, -314.79) mm, rotated rx -178.51 ry -54.99 rz -31.3 deg; joints [1.678, -25.384, 76.398, -254.001, 46.453, 293.461]
  MoveL 803 to (-309.2, 4.71, -314.5) mm, rotated rx -178.51 ry -54.99 rz -31.3 deg; joints [1.681, -25.408, 76.436, -253.985, 46.455, 293.441]
  MoveL 804 to (-309.12, 4.86, -314.2) mm, rotated rx -178.51 ry -54.99 rz -31.3 deg; joints [1.684, -25.431, 76.474, -253.968, 46.457, 293.421]
  MoveL 805 to (-309.04, 4.98, -313.91) mm, rotated rx -178.51 ry -54.99 rz -31.3 deg; joints [1.687, -25.453, 76.512, -253.952, 46.459, 293.4]
  MoveL 806 to (-308.98, 5.09, -313.62) mm, rotated rx -178.51 ry -54.99 rz -31.3 deg; joints [1.689, -25.475, 76.549, -253.935, 46.462, 293.378]
  MoveL 807 to (-308.88, 5.27, -313.03) mm, rotated rx -178.51 ry -54.99 rz -31.3 deg; joints [1.693, -25.516, 76.624, -253.901, 46.469, 293.333]
  MoveL 808 to (-308.82, 5.37, -312.58) mm, rotated rx -178.51 ry -54.99 rz -31.3 deg; joints [1.695, -25.545, 76.68, -253.874, 46.475, 293.298]
  MoveL 809 to (-308.79, 5.43, -312.23) mm, rotated rx -178.51 ry -54.99 rz -31.3 deg; joints [1.697, -25.568, 76.723, -253.854, 46.48, 293.269]
  MoveL 810 to (-308.76, 5.47, -311.88) mm, rotated rx -178.51 ry -54.99 rz -31.3 deg; joints [1.698, -25.589, 76.767, -253.832, 46.486, 293.239]
  MoveL 811 to (-308.75, 5.49, -311.54) mm, rotated rx -178.51 ry -54.99 rz -31.3 deg; joints [1.699, -25.61, 76.81, -253.811, 46.492, 293.209]
  MoveL 812 to (-308.75, 5.49, -311.19) mm, rotated rx -178.51 ry -54.99 rz -31.3 deg; joints [1.699, -25.63, 76.853, -253.79, 46.498, 293.179]
  MoveL 813 to (-308.75, 5.49, -5.24) mm, rotated rx -178.51 ry -54.99 rz -31.3 deg; joints [2.08, -39.256, 108.27, -239.531, 53.469, 271.712]
  MoveL 814 to (-308.75, 5.49, -2.45) mm, rotated rx -178.51 ry -54.99 rz -31.3 deg; joints [2.084, -39.356, 108.518, -239.432, 53.544, 271.552]
  MoveL 815 to (-308.76, 5.46, -2.07) mm, rotated rx -178.51 ry -54.99 rz -31.3 deg; joints [2.084, -39.368, 108.551, -239.419, 53.554, 271.53]
  MoveL 816 to (-308.79, 5.42, -1.7) mm, rotated rx -178.51 ry -54.99 rz -31.3 deg; joints [2.084, -39.379, 108.584, -239.405, 53.566, 271.506]
  MoveL 817 to (-308.83, 5.36, -1.32) mm, rotated rx -178.51 ry -54.99 rz -31.3 deg; joints [2.083, -39.388, 108.616, -239.392, 53.577, 271.482]
  MoveL 818 to (-308.88, 5.27, -0.95) mm, rotated rx -178.51 ry -54.99 rz -31.3 deg; joints [2.082, -39.397, 108.649, -239.378, 53.59, 271.457]
  MoveL 819 to (-308.93, 5.18, -0.63) mm, rotated rx -178.51 ry -54.99 rz -31.3 deg; joints [2.08, -39.403, 108.676, -239.366, 53.601, 271.435]
  MoveL 820 to (-308.99, 5.07, -0.3) mm, rotated rx -178.51 ry -54.99 rz -31.3 deg; joints [2.078, -39.409, 108.704, -239.354, 53.613, 271.411]
  MoveL 821 to (-309.06, 4.95, 0.02) mm, rotated rx -178.51 ry -54.99 rz -31.3 deg; joints [2.076, -39.413, 108.732, -239.342, 53.626, 271.387]
  MoveL 822 to (-309.15, 4.8, 0.35) mm, rotated rx -178.51 ry -54.99 rz -31.3 deg; joints [2.073, -39.416, 108.759, -239.33, 53.639, 271.362]
  MoveL 823 to (-309.24, 4.65, 0.64) mm, rotated rx -178.51 ry -54.99 rz -31.3 deg; joints [2.07, -39.418, 108.783, -239.319, 53.651, 271.339]
  MoveL 824 to (-309.33, 4.48, 0.93) mm, rotated rx -178.51 ry -54.99 rz -31.3 deg; joints [2.066, -39.419, 108.807, -239.308, 53.664, 271.315]
  MoveL 825 to (-309.44, 4.29, 1.22) mm, rotated rx -178.51 ry -54.99 rz -31.3 deg; joints [2.062, -39.418, 108.831, -239.297, 53.678, 271.29]
  MoveL 826 to (-309.57, 4.08, 1.51) mm, rotated rx -178.51 ry -54.99 rz -31.3 deg; joints [2.058, -39.416, 108.854, -239.286, 53.692, 271.264]
  MoveL 827 to (-309.75, 3.77, 1.87) mm, rotated rx -178.51 ry -54.99 rz -31.3 deg; joints [2.051, -39.412, 108.883, -239.272, 53.711, 271.23]
  MoveL 828 to (-309.92, 3.47, 2.18) mm, rotated rx -178.51 ry -54.99 rz -31.3 deg; joints [2.045, -39.405, 108.907, -239.26, 53.729, 271.199]
  MoveL 829 to (-310.1, 3.16, 2.45) mm, rotated rx -178.51 ry -54.99 rz -31.3 deg; joints [2.038, -39.397, 108.927, -239.249, 53.745, 271.17]
  MoveL 830 to (-310.27, 2.86, 2.68) mm, rotated rx -178.51 ry -54.99 rz -31.3 deg; joints [2.032, -39.388, 108.944, -239.239, 53.76, 271.143]
  MoveL 831 to (-310.39, 2.66, 2.81) mm, rotated rx -178.51 ry -54.99 rz -31.3 deg; joints [2.027, -39.381, 108.953, -239.234, 53.77, 271.127]
  MoveL 832 to (-310.51, 2.46, 2.93) mm, rotated rx -178.51 ry -54.99 rz -31.3 deg; joints [2.023, -39.374, 108.962, -239.229, 53.779, 271.111]
  MoveL 833 to (-310.74, 2.06, 3.14) mm, rotated rx -178.51 ry -54.99 rz -31.3 deg; joints [2.014, -39.358, 108.976, -239.22, 53.797, 271.082]
  MoveL 834 to (-310.97, 1.66, 3.31) mm, rotated rx -178.51 ry -54.99 rz -31.3 deg; joints [2.005, -39.341, 108.986, -239.212, 53.814, 271.054]
  MoveL 835 to (-311.2, 1.25, 3.44) mm, rotated rx -178.51 ry -54.99 rz -31.3 deg; joints [1.996, -39.322, 108.993, -239.206, 53.83, 271.029]
  MoveL 836 to (-311.44, 0.85, 3.53) mm, rotated rx -178.51 ry -54.99 rz -31.3 deg; joints [1.987, -39.302, 108.996, -239.201, 53.845, 271.006]
  MoveL 837 to (-311.67, 0.44, 3.59) mm, rotated rx -178.51 ry -54.99 rz -31.3 deg; joints [1.977, -39.28, 108.996, -239.197, 53.858, 270.985]
  MoveL 838 to (-311.85, 0.14, 3.6) mm, rotated rx -178.51 ry -54.99 rz -31.3 deg; joints [1.97, -39.264, 108.994, -239.195, 53.868, 270.971]
  MoveL 839 to (-312.02, -0.16, 3.61) mm, rotated rx -178.51 ry -54.99 rz -31.3 deg; joints [1.963, -39.246, 108.991, -239.194, 53.877, 270.958]
  MoveL 840 to (-313.77, -3.18, 3.61) mm, rotated rx -178.51 ry -54.99 rz -31.3 deg; joints [1.894, -39.072, 108.956, -239.181, 53.969, 270.825]
  MoveL 841 to (-314.12, -3.78, 3.58) mm, rotated rx -178.51 ry -54.99 rz -31.3 deg; joints [1.88, -39.036, 108.946, -239.179, 53.987, 270.8]
  MoveL 842 to (-314.47, -4.39, 3.49) mm, rotated rx -178.51 ry -54.99 rz -31.3 deg; joints [1.866, -38.998, 108.931, -239.18, 54.003, 270.779]
  MoveL 843 to (-318.67, -11.63, 2.16) mm, rotated rx -178.51 ry -54.99 rz -31.3 deg; joints [1.697, -38.531, 108.723, -239.199, 54.185, 270.54]
  MoveL 844 to (-320.06, -14.04, 1.71) mm, rotated rx -178.51 ry -54.99 rz -31.3 deg; joints [1.641, -38.375, 108.652, -239.206, 54.245, 270.463]
  MoveL 845 to (-320.24, -14.34, 1.62) mm, rotated rx -178.51 ry -54.99 rz -31.3 deg; joints [1.634, -38.355, 108.64, -239.208, 54.251, 270.455]
  MoveL 846 to (-320.41, -14.63, 1.52) mm, rotated rx -178.51 ry -54.99 rz -31.3 deg; joints [1.627, -38.334, 108.627, -239.211, 54.257, 270.448]
  MoveL 847 to (-320.58, -14.93, 1.39) mm, rotated rx -178.51 ry -54.99 rz -31.3 deg; joints [1.62, -38.312, 108.612, -239.214, 54.262, 270.443]
  MoveL 848 to (-320.75, -15.22, 1.24) mm, rotated rx -178.51 ry -54.99 rz -31.3 deg; joints [1.613, -38.29, 108.594, -239.219, 54.267, 270.439]
  MoveL 849 to (-320.92, -15.52, 1.06) mm, rotated rx -178.51 ry -54.99 rz -31.3 deg; joints [1.606, -38.266, 108.575, -239.224, 54.271, 270.437]
  MoveL 850 to (-321.09, -15.82, 0.85) mm, rotated rx -178.51 ry -54.99 rz -31.3 deg; joints [1.599, -38.242, 108.553, -239.23, 54.274, 270.436]
  MoveL 851 to (-321.26, -16.11, 0.62) mm, rotated rx -178.51 ry -54.99 rz -31.3 deg; joints [1.592, -38.217, 108.528, -239.237, 54.276, 270.437]
  MoveL 852 to (-321.43, -16.41, 0.35) mm, rotated rx -178.51 ry -54.99 rz -31.3 deg; joints [1.585, -38.19, 108.5, -239.245, 54.278, 270.44]
  MoveL 853 to (-321.46, -16.46, 0.3) mm, rotated rx -178.51 ry -54.99 rz -31.3 deg; joints [1.584, -38.185, 108.495, -239.247, 54.278, 270.44]
  MoveC 854 to (-321.99, -17.38, 0.01) mm, rotated rx -178.51 ry -54.99 rz -31.3 deg; joints [1.562, -38.122, 108.457, -239.254, 54.297, 270.418] to (-322.44, -18.14, 0.66) mm, rotated rx -178.51 ry -54.99 rz -31.3 deg; joints [1.545, -38.1, 108.504, -239.229, 54.338, 270.348]
  MoveL 855 to (-322.44, -18.14, 0.66) mm, rotated rx -178.51 ry -54.99 rz -31.3 deg; joints [1.545, -38.1, 108.504, -239.229, 54.338, 270.348]
  MoveL 856 to (-323.43, -19.85, 4.32) mm, rotated rx -178.51 ry -54.99 rz -31.3 deg; joints [1.51, -38.127, 108.806, -239.098, 54.488, 270.066]
  MoveL 857 to (-324.83, -19.73, 5.44) mm, rotated rx -178.51 ry -54.99 rz -31.3 deg; joints [1.455, -38.173, 108.91, -239.121, 54.533, 270.016]
  Set speed (200.0 mm/s)
  MoveL 858 to (-336.31, -13.08, 5.44) mm, rotated rx -178.51 ry -54.99 rz -31.3 deg; joints [0.993, -38.571, 109.031, -239.783, 54.525, 270.405]
  Print: /'Parallel1'
  Call SetTool(1)
  Set speed (200.0 mm/s)
  MoveL 859 to (-340.11, 16.27, -316.36) mm, rotated rx -178.51 ry -54.99 rz -31.3 deg; joints [0.664, -25.88, 76.445, -255.353, 46.952, 294.288]
  MoveL 860 to (-319.42, 4.29, -316.36) mm, rotated rx -178.51 ry -54.99 rz -31.3 deg; joints [1.344, -25.296, 76.234, -254.383, 46.634, 293.641]
  Set speed (100.0 mm/s)
  MoveL 861 to (-318.78, 3.92, -316.36) mm, rotated rx -178.51 ry -54.99 rz -31.3 deg; joints [1.365, -25.278, 76.227, -254.354, 46.624, 293.621]
  MoveC 862 to (-318.01, 3.47, -315.99) mm, rotated rx -178.51 ry -54.99 rz -31.3 deg; joints [1.391, -25.277, 76.265, -254.295, 46.619, 293.564] to (-317.69, 3.28, -315.09) mm, rotated rx -178.51 ry -54.99 rz -31.3 deg; joints [1.402, -25.318, 76.372, -254.224, 46.63, 293.474]
  MoveL 863 to (-317.69, 3.28, -315.09) mm, rotated rx -178.51 ry -54.99 rz -31.3 deg; joints [1.402, -25.318, 76.372, -254.224, 46.63, 293.474]
  MoveL 864 to (-317.69, 3.28, 0.74) mm, rotated rx -178.51 ry -54.99 rz -31.3 deg; joints [1.732, -39.351, 108.8, -239.627, 53.796, 271.324]
  MoveL 865 to (-317.74, 3.32, 1.02) mm, rotated rx -178.51 ry -54.99 rz -31.3 deg; joints [1.73, -39.362, 108.825, -239.62, 53.804, 271.31]
  MoveL 866 to (-317.8, 3.35, 1.3) mm, rotated rx -178.51 ry -54.99 rz -31.3 deg; joints [1.728, -39.374, 108.85, -239.614, 53.811, 271.296]
  MoveL 867 to (-317.8, 3.35, 2.99) mm, rotated rx -178.51 ry -54.99 rz -31.3 deg; joints [1.73, -39.434, 109, -239.555, 53.856, 271.2]
  MoveC 868 to (-318.08, 2.86, 4.33) mm, rotated rx -178.51 ry -54.99 rz -31.3 deg; joints [1.721, -39.454, 109.114, -239.506, 53.906, 271.102] to (-318.75, 1.7, 4.89) mm, rotated rx -178.51 ry -54.99 rz -31.3 deg; joints [1.695, -39.407, 109.149, -239.481, 53.956, 271.018]
  MoveL 869 to (-318.75, 1.7, 4.89) mm, rotated rx -178.51 ry -54.99 rz -31.3 deg; joints [1.695, -39.407, 109.149, -239.481, 53.956, 271.018]
  MoveL 870 to (-320.03, -0.5, 4.89) mm, rotated rx -178.51 ry -54.99 rz -31.3 deg; joints [1.644, -39.279, 109.123, -239.472, 54.023, 270.922]
  MoveC 871 to (-320.7, -1.66, 4.33) mm, rotated rx -178.51 ry -54.99 rz -31.3 deg; joints [1.617, -39.192, 109.06, -239.487, 54.043, 270.902] to (-320.98, -2.15, 2.99) mm, rotated rx -178.51 ry -54.99 rz -31.3 deg; joints [1.604, -39.117, 108.935, -239.531, 54.022, 270.958]
  MoveL 872 to (-320.98, -2.15, 2.99) mm, rotated rx -178.51 ry -54.99 rz -31.3 deg; joints [1.604, -39.117, 108.935, -239.531, 54.022, 270.958]
  MoveL 873 to (-320.92, -2.18, 2.71) mm, rotated rx -178.51 ry -54.99 rz -31.3 deg; joints [1.606, -39.105, 108.91, -239.538, 54.014, 270.972]
  MoveL 874 to (-320.87, -2.21, 2.43) mm, rotated rx -178.51 ry -54.99 rz -31.3 deg; joints [1.608, -39.093, 108.884, -239.544, 54.007, 270.986]
  MoveL 875 to (-320.87, -2.21, -317.02) mm, rotated rx -178.51 ry -54.99 rz -31.3 deg; joints [1.297, -24.953, 76.064, -254.271, 46.709, 293.423]
  MoveL 876 to (-320.92, -2.18, -317.3) mm, rotated rx -178.51 ry -54.99 rz -31.3 deg; joints [1.295, -24.939, 76.029, -254.291, 46.705, 293.45]
  MoveL 877 to (-320.98, -2.15, -317.58) mm, rotated rx -178.51 ry -54.99 rz -31.3 deg; joints [1.293, -24.924, 75.995, -254.311, 46.701, 293.477]
  MoveL 878 to (-320.98, -2.15, -317.58) mm, rotated rx -178.51 ry -54.99 rz -31.3 deg; joints [1.293, -24.924, 75.995, -254.311, 46.701, 293.477]
  MoveC 879 to (-321.26, -2.63, -318.92) mm, rotated rx -178.51 ry -54.99 rz -31.3 deg; joints [1.283, -24.826, 75.822, -254.388, 46.687, 293.578] to (-321.94, -3.79, -319.48) mm, rotated rx -178.51 ry -54.99 rz -31.3 deg; joints [1.26, -24.739, 75.737, -254.408, 46.701, 293.582]
  MoveL 880 to (-321.94, -3.79, -319.48) mm, rotated rx -178.51 ry -54.99 rz -31.3 deg; joints [1.26, -24.739, 75.737, -254.408, 46.701, 293.582]
  MoveL 881 to (-323.21, -5.99, -319.48) mm, rotated rx -178.51 ry -54.99 rz -31.3 deg; joints [1.219, -24.636, 75.707, -254.38, 46.746, 293.494]
  MoveC 882 to (-323.88, -7.16, -318.92) mm, rotated rx -178.51 ry -54.99 rz -31.3 deg; joints [1.198, -24.613, 75.761, -254.33, 46.779, 293.397] to (-324.16, -7.64, -317.58) mm, rotated rx -178.51 ry -54.99 rz -31.3 deg; joints [1.189, -24.666, 75.922, -254.24, 46.813, 293.256]
  MoveL 883 to (-324.16, -7.64, -317.58) mm, rotated rx -178.51 ry -54.99 rz -31.3 deg; joints [1.189, -24.666, 75.922, -254.24, 46.813, 293.256]
  MoveL 884 to (-324.11, -7.67, -317.3) mm, rotated rx -178.51 ry -54.99 rz -31.3 deg; joints [1.192, -24.68, 75.956, -254.22, 46.818, 293.229]
  MoveL 885 to (-324.11, -7.67, -317.3) mm, rotated rx -178.51 ry -54.99 rz -31.3 deg; joints [1.192, -24.68, 75.956, -254.22, 46.818, 293.229]
  MoveL 886 to (-324.05, -7.7, -317.02) mm, rotated rx -178.51 ry -54.99 rz -31.3 deg; joints [1.194, -24.694, 75.99, -254.2, 46.822, 293.203]
  MoveL 887 to (-324.05, -7.7, 1.46) mm, rotated rx -178.51 ry -54.99 rz -31.3 deg; joints [1.48, -38.741, 108.731, -239.556, 54.146, 270.801]
  MoveC 888 to (-324.37, -7.52, 2.36) mm, rotated rx -178.51 ry -54.99 rz -31.3 deg; joints [1.468, -38.783, 108.814, -239.543, 54.169, 270.761] to (-325.15, -7.07, 2.73) mm, rotated rx -178.51 ry -54.99 rz -31.3 deg; joints [1.437, -38.823, 108.855, -239.575, 54.179, 270.766]
  MoveL 889 to (-325.15, -7.07, 2.73) mm, rotated rx -178.51 ry -54.99 rz -31.3 deg; joints [1.437, -38.823, 108.855, -239.575, 54.179, 270.766]
  Set speed (200.0 mm/s)
  MoveL 890 to (-346.48, 5.29, 2.73) mm, rotated rx -178.51 ry -54.99 rz -31.3 deg; joints [0.58, -39.554, 109.057, -240.817, 54.174, 271.514]
  MoveL 891 to (-346.48, 5.29, 2.73) mm, rotated rx -178.51 ry -54.99 rz -31.3 deg; joints [0.58, -39.554, 109.057, -240.817, 54.174, 271.514]
